  Set speed (30.0 mm/s)
  Call Extruder(0.767)
  MoveL 6356 to (509.32, 509.32, 13.5) mm, rotated rx 0 ry 90 rz 0 deg; joints [-12.669, -27.494, 110.087, -16.732, -82.041, 51.355]
  MoveL 6357 to (509.44, 509.44, 13.5) mm, rotated rx 0 ry 90 rz 0 deg; joints [-12.677, -27.491, 110.069, -16.741, -82.027, 51.361]
  Set speed (120.0 mm/s)
  MoveL 6358 to (507.39, 502.51, 13.5) mm, rotated rx 0 ry 90 rz 0 deg; joints [-12.094, -27.562, 110.499, -16.138, -82.35, 51.187]
  Set speed (30.0 mm/s)
  Call Extruder(0.280)
  MoveL 6359 to (500.58, 509.32, 13.5) mm, rotated rx 0 ry 90 rz 0 deg; joints [-12.847, -27.665, 111.134, -16.878, -82.886, 51.121]
  Set speed (120.0 mm/s)
  MoveL 6360 to (499.42, 509.32, 13.5) mm, rotated rx 0 ry 90 rz 0 deg; joints [-12.872, -27.687, 111.272, -16.898, -82.998, 51.089]
  Set speed (30.0 mm/s)
  Call Extruder(0.360)
  MoveL 6361 to (490.68, 500.58, 13.5) mm, rotated rx 0 ry 90 rz 0 deg; joints [-12.247, -27.877, 112.54, -16.235, -84.012, 50.718]
  Set speed (120.0 mm/s)
  MoveL 6362 to (490.68, 499.42, 13.5) mm, rotated rx 0 ry 90 rz 0 deg; joints [-12.139, -27.882, 112.569, -16.126, -84.034, 50.702]
  Set speed (30.0 mm/s)
  Call Extruder(0.281)
  MoveL 6363 to (497.52, 492.58, 13.5) mm, rotated rx 0 ry 90 rz 0 deg; joints [-11.373, -27.787, 111.927, -15.372, -83.486, 50.779]
  MoveL 6364 to (497.64, 492.46, 13.5) mm, rotated rx 0 ry 90 rz 0 deg; joints [-11.359, -27.786, 111.915, -15.359, -83.476, 50.78]
  Set speed (120.0 mm/s)
  MoveL 6365 to (499.02, 491.08, 13.5) mm, rotated rx 0 ry 90 rz 0 deg; joints [-11.207, -27.766, 111.784, -15.208, -83.364, 50.795]
  Set speed (30.0 mm/s)
  Call Extruder(0.016)
  MoveL 6366 to (499.42, 490.68, 13.5) mm, rotated rx 0 ry 90 rz 0 deg; joints [-11.163, -27.76, 111.745, -15.165, -83.331, 50.799]
  Set speed (120.0 mm/s)
  MoveL 6367 to (500.44, 492.33, 13.5) mm, rotated rx 0 ry 90 rz 0 deg; joints [-11.296, -27.735, 111.584, -15.303, -83.203, 50.849]
  Set speed (1000.0 mm/s)
  MoveL 6368 to (502.48, 492.58, 13.5) mm, rotated rx 0 ry 90 rz 0 deg; joints [-11.282, -27.697, 111.335, -15.296, -82.999, 50.903]
  Set speed (30.0 mm/s)
  Call Extruder(0.202)
  MoveL 6369 to (507.39, 497.49, 13.5) mm, rotated rx 0 ry 90 rz 0 deg; joints [-11.639, -27.583, 110.626, -15.676, -82.436, 51.104]
  MoveL 6370 to (507.51, 497.61, 13.5) mm, rotated rx 0 ry 90 rz 0 deg; joints [-11.648, -27.58, 110.608, -15.685, -82.422, 51.109]
  Set speed (120.0 mm/s)
  MoveL 6371 to (508.52, 498.62, 13.5) mm, rotated rx 0 ry 90 rz 0 deg; joints [-11.72, -27.556, 110.461, -15.763, -82.307, 51.151]
  Set speed (30.0 mm/s)
  Call Extruder(0.033)
  MoveL 6372 to (509.32, 499.42, 13.5) mm, rotated rx 0 ry 90 rz 0 deg; joints [-11.777, -27.537, 110.345, -15.824, -82.216, 51.185]
  Set speed (120.0 mm/s)
  MoveL 6373 to (507.64, 498.37, 13.5) mm, rotated rx 0 ry 90 rz 0 deg; joints [-11.714, -27.575, 110.573, -15.753, -82.397, 51.125]
  Set speed (1000.0 mm/s)
  MoveL 6374 to (507.64, 495.81, 13.5) mm, rotated rx 0 ry 90 rz 0 deg; joints [-11.481, -27.585, 110.637, -15.517, -82.44, 51.083]
  Set speed (1000.0 mm/s)
  MoveL 6375 to (509.32, 490.68, 13.5) mm, rotated rx 0 ry 90 rz 0 deg; joints [-10.985, -27.572, 110.557, -15.019, -82.36, 51.042]
  Set speed (30.0 mm/s)
  Call Extruder(0.767)
  MoveL 6376 to (490.68, 509.32, 13.5) mm, rotated rx 0 ry 90 rz 0 deg; joints [-13.056, -27.844, 112.308, -17.054, -83.844, 50.849]
  MoveL 6377 to (490.56, 509.44, 13.5) mm, rotated rx 0 ry 90 rz 0 deg; joints [-13.07, -27.845, 112.319, -17.068, -83.854, 50.848]
  Set speed (120.0 mm/s)
  MoveL 6378 to (502.97, 492.37, 13.5) mm, rotated rx 0 ry 90 rz 0 deg; joints [-11.253, -27.688, 111.281, -15.269, -82.954, 50.912]
  Set speed (1000.0 mm/s)
  MoveL 6379 to (502.9, 492.3, 13.5) mm, rotated rx 0 ry 90 rz 0 deg; joints [-11.248, -27.69, 111.291, -15.263, -82.962, 50.91]
  Set speed (15.0 mm/s)
  Call Extruder(0.010)
  MoveL 6380 to (502.9, 491.95, 13.5) mm, rotated rx 0 ry 90 rz 0 deg; joints [-11.216, -27.691, 111.299, -15.231, -82.968, 50.904]
  Call Extruder(0.035)
  MoveL 6381 to (502.9, 490.75, 13.5) mm, rotated rx 0 ry 90 rz 0 deg; joints [-11.106, -27.696, 111.328, -15.119, -82.988, 50.886]
  Call Extruder(0.010)
  MoveL 6382 to (502.9, 490.4, 13.5) mm, rotated rx 0 ry 90 rz 0 deg; joints [-11.074, -27.697, 111.336, -15.087, -82.994, 50.881]
  Call Extruder(0.007)
  MoveL 6383 to (503.25, 490.4, 13.5) mm, rotated rx 0 ry 90 rz 0 deg; joints [-11.068, -27.69, 111.294, -15.081, -82.96, 50.889]
  Call Extruder(0.185)
  MoveL 6384 to (509.6, 490.4, 13.5) mm, rotated rx 0 ry 90 rz 0 deg; joints [-10.955, -27.568, 110.53, -14.989, -82.337, 51.044]
  Call Extruder(0.158)
  MoveL 6385 to (509.6, 495.84, 13.5) mm, rotated rx 0 ry 90 rz 0 deg; joints [-11.448, -27.546, 110.4, -15.49, -82.249, 51.132]
  Call Extruder(0.056)
  MoveL 6386 to (507.67, 495.84, 13.5) mm, rotated rx 0 ry 90 rz 0 deg; joints [-11.483, -27.584, 110.632, -15.519, -82.437, 51.084]
  Call Extruder(0.063)
  MoveL 6387 to (507.67, 497.99, 13.5) mm, rotated rx 0 ry 90 rz 0 deg; joints [-11.679, -27.576, 110.579, -15.718, -82.4, 51.119]
  Call Extruder(0.010)
  MoveL 6388 to (507.67, 498.34, 13.5) mm, rotated rx 0 ry 90 rz 0 deg; joints [-11.711, -27.574, 110.571, -15.75, -82.394, 51.125]
  Call Extruder(0.007)
  MoveL 6389 to (508.02, 498.34, 13.5) mm, rotated rx 0 ry 90 rz 0 deg; joints [-11.704, -27.567, 110.528, -15.745, -82.36, 51.134]
  Call Extruder(0.036)
  MoveL 6390 to (509.25, 498.34, 13.5) mm, rotated rx 0 ry 90 rz 0 deg; joints [-11.681, -27.543, 110.38, -15.726, -82.241, 51.165]
  Call Extruder(0.010)
  MoveL 6391 to (509.6, 498.34, 13.5) mm, rotated rx 0 ry 90 rz 0 deg; joints [-11.675, -27.536, 110.338, -15.721, -82.206, 51.174]
  Call Extruder(0.007)
  MoveL 6392 to (509.6, 498.69, 13.5) mm, rotated rx 0 ry 90 rz 0 deg; joints [-11.706, -27.534, 110.329, -15.753, -82.201, 51.18]
  Call Extruder(0.050)
  MoveL 6393 to (509.6, 500.4, 13.5) mm, rotated rx 0 ry 90 rz 0 deg; joints [-11.86, -27.527, 110.287, -15.91, -82.171, 51.208]
  Call Extruder(0.010)
  MoveL 6394 to (509.6, 500.75, 13.5) mm, rotated rx 0 ry 90 rz 0 deg; joints [-11.892, -27.526, 110.278, -15.942, -82.165, 51.214]
  Call Extruder(0.007)
  MoveL 6395 to (509.25, 500.75, 13.5) mm, rotated rx 0 ry 90 rz 0 deg; joints [-11.898, -27.533, 110.32, -15.947, -82.199, 51.205]
  Call Extruder(0.036)
  MoveL 6396 to (508.02, 500.75, 13.5) mm, rotated rx 0 ry 90 rz 0 deg; joints [-11.922, -27.557, 110.468, -15.966, -82.319, 51.174]
  Call Extruder(0.010)
  MoveL 6397 to (507.67, 500.75, 13.5) mm, rotated rx 0 ry 90 rz 0 deg; joints [-11.928, -27.564, 110.51, -15.971, -82.353, 51.165]
  Call Extruder(0.007)
  MoveL 6398 to (507.67, 501.1, 13.5) mm, rotated rx 0 ry 90 rz 0 deg; joints [-11.96, -27.563, 110.501, -16.003, -82.347, 51.17]
  Call Extruder(0.062)
  MoveL 6399 to (507.67, 503.24, 13.5) mm, rotated rx 0 ry 90 rz 0 deg; joints [-12.154, -27.554, 110.446, -16.201, -82.31, 51.206]
  Call Extruder(0.056)
  MoveL 6400 to (509.6, 503.24, 13.5) mm, rotated rx 0 ry 90 rz 0 deg; joints [-12.117, -27.515, 110.214, -16.171, -82.122, 51.257]
  Call Extruder(0.185)
  MoveL 6401 to (509.6, 509.6, 13.5) mm, rotated rx 0 ry 90 rz 0 deg; joints [-12.688, -27.487, 110.045, -16.753, -82.009, 51.368]
  Call Extruder(0.559)
  MoveL 6402 to (490.4, 509.6, 13.5) mm, rotated rx 0 ry 90 rz 0 deg; joints [-13.088, -27.848, 112.333, -17.086, -83.866, 50.846]
  MoveL 6403 to (490.4, 490.4, 13.5) mm, rotated rx 0 ry 90 rz 0 deg; joints [-11.303, -27.917, 112.824, -15.28, -84.223, 50.569]
  Call Extruder(0.161)
  MoveL 6404 to (495.93, 490.4, 13.5) mm, rotated rx 0 ry 90 rz 0 deg; joints [-11.201, -27.823, 112.167, -15.192, -83.678, 50.708]
  Call Extruder(0.010)
  MoveL 6405 to (496.28, 490.4, 13.5) mm, rotated rx 0 ry 90 rz 0 deg; joints [-11.194, -27.817, 112.126, -15.187, -83.644, 50.717]
  Call Extruder(0.007)
  MoveL 6406 to (496.28, 490.75, 13.5) mm, rotated rx 0 ry 90 rz 0 deg; joints [-11.227, -27.816, 112.118, -15.22, -83.638, 50.722]
  Call Extruder(0.035)
  MoveL 6407 to (496.28, 491.95, 13.5) mm, rotated rx 0 ry 90 rz 0 deg; joints [-11.338, -27.812, 112.089, -15.332, -83.618, 50.739]
  Call Extruder(0.010)
  MoveL 6408 to (496.28, 492.3, 13.5) mm, rotated rx 0 ry 90 rz 0 deg; joints [-11.37, -27.81, 112.081, -15.365, -83.612, 50.744]
  Call Extruder(0.007)
  MoveL 6409 to (496.63, 492.3, 13.5) mm, rotated rx 0 ry 90 rz 0 deg; joints [-11.364, -27.804, 112.039, -15.36, -83.577, 50.753]
  Call Extruder(0.061)
  MoveL 6410 to (498.74, 492.3, 13.5) mm, rotated rx 0 ry 90 rz 0 deg; joints [-11.325, -27.767, 111.788, -15.327, -83.37, 50.806]
  Call Extruder(0.055)
  MoveL 6411 to (498.74, 490.4, 13.5) mm, rotated rx 0 ry 90 rz 0 deg; joints [-11.149, -27.773, 111.833, -15.149, -83.402, 50.778]
  Call Extruder(0.050)
  MoveL 6412 to (500.47, 490.4, 13.5) mm, rotated rx 0 ry 90 rz 0 deg; joints [-11.118, -27.742, 111.627, -15.123, -83.233, 50.821]
  Call Extruder(0.055)
  MoveL 6413 to (500.47, 492.3, 13.5) mm, rotated rx 0 ry 90 rz 0 deg; joints [-11.293, -27.735, 111.581, -15.3, -83.201, 50.849]
  Call Extruder(0.060)
  MoveL 6414 to (502.55, 492.3, 13.5) mm, rotated rx 0 ry 90 rz 0 deg; joints [-11.255, -27.696, 111.333, -15.268, -82.997, 50.901]
  Call Extruder(0.007)
  MoveL 6415 to (502.9, 492.3, 13.5) mm, rotated rx 0 ry 90 rz 0 deg; joints [-11.248, -27.69, 111.291, -15.263, -82.962, 50.91]
  Set speed (120.0 mm/s)
  MoveL 6416 to (502.9, 491.95, 13.5) mm, rotated rx 0 ry 90 rz 0 deg; joints [-11.216, -27.691, 111.299, -15.231, -82.968, 50.904]
  Set speed (1000.0 mm/s)
  MoveL 6417 to (502.9, 491.9, 13.5) mm, rotated rx 0 ry 90 rz 0 deg; joints [-11.212, -27.691, 111.3, -15.226, -82.969, 50.903]
  Set speed (1000.0 mm/s)
  MoveL 6418 to (503.6, 491.9, 13.5) mm, rotated rx 0 ry 90 rz 0 deg; joints [-11.199, -27.678, 111.216, -15.216, -82.901, 50.921]
  Set speed (1000.0 mm/s)
  MoveL 6419 to (496.25, 492.33, 13.5) mm, rotated rx 0 ry 90 rz 0 deg; joints [-11.373, -27.811, 112.083, -15.368, -83.614, 50.744]
  Set speed (1000.0 mm/s)
  MoveL 6420 to (490.68, 490.68, 13.5) mm, rotated rx 0 ry 90 rz 0 deg; joints [-11.324, -27.912, 112.784, -15.302, -84.191, 50.58]
  Set speed (1000.0 mm/s)
  MoveL 6421 to (490.68, 490.68, 13.6) mm, rotated rx 0 ry 90 rz 0 deg; joints [-11.324, -27.923, 112.789, -15.302, -84.185, 50.581]
  Set speed (30.0 mm/s)
  Call Extruder(0.767)
  MoveL 6422 to (509.32, 509.32, 13.6) mm, rotated rx 0 ry 90 rz 0 deg; joints [-12.669, -27.504, 110.092, -16.732, -82.036, 51.357]
  MoveL 6423 to (509.44, 509.44, 13.6) mm, rotated rx 0 ry 90 rz 0 deg; joints [-12.677, -27.501, 110.074, -16.741, -82.022, 51.362]
  Set speed (120.0 mm/s)
  MoveL 6424 to (507.39, 502.51, 13.6) mm, rotated rx 0 ry 90 rz 0 deg; joints [-12.094, -27.573, 110.504, -16.138, -82.345, 51.188]
  Set speed (30.0 mm/s)
  Call Extruder(0.280)
  MoveL 6425 to (500.58, 509.32, 13.6) mm, rotated rx 0 ry 90 rz 0 deg; joints [-12.847, -27.676, 111.139, -16.878, -82.88, 51.122]
  Set speed (120.0 mm/s)
  MoveL 6426 to (499.42, 509.32, 13.6) mm, rotated rx 0 ry 90 rz 0 deg; joints [-12.872, -27.698, 111.277, -16.899, -82.992, 51.091]
  Set speed (30.0 mm/s)
  Call Extruder(0.360)
  MoveL 6427 to (490.68, 500.58, 13.6) mm, rotated rx 0 ry 90 rz 0 deg; joints [-12.247, -27.888, 112.545, -16.235, -84.007, 50.72]
  Set speed (120.0 mm/s)
  MoveL 6428 to (490.68, 499.42, 13.6) mm, rotated rx 0 ry 90 rz 0 deg; joints [-12.139, -27.892, 112.575, -16.126, -84.028, 50.703]
  Set speed (30.0 mm/s)
  Call Extruder(0.281)
  MoveL 6429 to (497.52, 492.58, 13.6) mm, rotated rx 0 ry 90 rz 0 deg; joints [-11.373, -27.798, 111.932, -15.372, -83.48, 50.781]
  MoveL 6430 to (497.64, 492.46, 13.6) mm, rotated rx 0 ry 90 rz 0 deg; joints [-11.36, -27.796, 111.92, -15.359, -83.47, 50.782]
  Set speed (120.0 mm/s)
  MoveL 6431 to (498.96, 491.14, 13.6) mm, rotated rx 0 ry 90 rz 0 deg; joints [-11.213, -27.777, 111.794, -15.215, -83.363, 50.796]
  Set speed (30.0 mm/s)
  Call Extruder(0.019)
  MoveL 6432 to (499.42, 490.68, 13.6) mm, rotated rx 0 ry 90 rz 0 deg; joints [-11.163, -27.771, 111.751, -15.165, -83.326, 50.8]
  Set speed (120.0 mm/s)
  MoveL 6433 to (500.51, 492.33, 13.6) mm, rotated rx 0 ry 90 rz 0 deg; joints [-11.295, -27.745, 111.582, -15.302, -83.191, 50.852]
  Set speed (1000.0 mm/s)
  MoveL 6434 to (502.48, 492.58, 13.6) mm, rotated rx 0 ry 90 rz 0 deg; joints [-11.282, -27.707, 111.34, -15.296, -82.994, 50.905]
  Set speed (30.0 mm/s)
  Call Extruder(0.202)
  MoveL 6435 to (507.39, 497.49, 13.6) mm, rotated rx 0 ry 90 rz 0 deg; joints [-11.639, -27.594, 110.631, -15.676, -82.431, 51.105]
  MoveL 6436 to (507.51, 497.61, 13.6) mm, rotated rx 0 ry 90 rz 0 deg; joints [-11.648, -27.591, 110.613, -15.685, -82.417, 51.11]
  Set speed (120.0 mm/s)
  MoveL 6437 to (508.46, 498.57, 13.6) mm, rotated rx 0 ry 90 rz 0 deg; joints [-11.716, -27.568, 110.475, -15.759, -82.308, 51.15]
  Set speed (30.0 mm/s)
  Call Extruder(0.035)
  MoveL 6438 to (509.32, 499.42, 13.6) mm, rotated rx 0 ry 90 rz 0 deg; joints [-11.777, -27.547, 110.35, -15.824, -82.21, 51.186]
  Set speed (120.0 mm/s)
  MoveL 6439 to (507.64, 498.31, 13.6) mm, rotated rx 0 ry 90 rz 0 deg; joints [-11.709, -27.585, 110.58, -15.748, -82.392, 51.125]
  Set speed (1000.0 mm/s)
  MoveL 6440 to (507.64, 495.75, 13.6) mm, rotated rx 0 ry 90 rz 0 deg; joints [-11.476, -27.596, 110.643, -15.511, -82.436, 51.083]
  Set speed (1000.0 mm/s)
  MoveL 6441 to (509.32, 490.68, 13.6) mm, rotated rx 0 ry 90 rz 0 deg; joints [-10.985, -27.583, 110.562, -15.019, -82.355, 51.043]
  Set speed (30.0 mm/s)
  Call Extruder(0.767)
  MoveL 6442 to (490.68, 509.32, 13.6) mm, rotated rx 0 ry 90 rz 0 deg; joints [-13.056, -27.854, 112.313, -17.055, -83.839, 50.851]
  MoveL 6443 to (490.56, 509.44, 13.6) mm, rotated rx 0 ry 90 rz 0 deg; joints [-13.07, -27.856, 112.325, -17.068, -83.848, 50.849]
  Set speed (120.0 mm/s)
  MoveL 6444 to (503.03, 492.37, 13.6) mm, rotated rx 0 ry 90 rz 0 deg; joints [-11.252, -27.698, 111.278, -15.268, -82.943, 50.915]
  Set speed (1000.0 mm/s)
  MoveL 6445 to (502.96, 492.3, 13.6) mm, rotated rx 0 ry 90 rz 0 deg; joints [-11.247, -27.699, 111.288, -15.262, -82.951, 50.913]
  Set speed (15.0 mm/s)
  Call Extruder(0.010)
  MoveL 6446 to (502.96, 491.95, 13.6) mm, rotated rx 0 ry 90 rz 0 deg; joints [-11.215, -27.701, 111.297, -15.23, -82.957, 50.907]
  Call Extruder(0.035)
  MoveL 6447 to (502.96, 490.75, 13.6) mm, rotated rx 0 ry 90 rz 0 deg; joints [-11.105, -27.705, 111.325, -15.118, -82.977, 50.889]
  Call Extruder(0.010)
  MoveL 6448 to (502.96, 490.4, 13.6) mm, rotated rx 0 ry 90 rz 0 deg; joints [-11.073, -27.706, 111.333, -15.086, -82.983, 50.884]
  Call Extruder(0.007)
  MoveL 6449 to (503.31, 490.4, 13.6) mm, rotated rx 0 ry 90 rz 0 deg; joints [-11.067, -27.7, 111.291, -15.081, -82.948, 50.892]
  Call Extruder(0.183)
  MoveL 6450 to (509.6, 490.4, 13.6) mm, rotated rx 0 ry 90 rz 0 deg; joints [-10.955, -27.578, 110.535, -14.989, -82.332, 51.046]
  Call Extruder(0.156)
  MoveL 6451 to (509.6, 495.78, 13.6) mm, rotated rx 0 ry 90 rz 0 deg; joints [-11.442, -27.557, 110.407, -15.485, -82.244, 51.133]
  Call Extruder(0.056)
  MoveL 6452 to (507.67, 495.78, 13.6) mm, rotated rx 0 ry 90 rz 0 deg; joints [-11.478, -27.595, 110.639, -15.514, -82.433, 51.084]
  Call Extruder(0.063)
  MoveL 6453 to (507.67, 497.94, 13.6) mm, rotated rx 0 ry 90 rz 0 deg; joints [-11.674, -27.586, 110.586, -15.713, -82.396, 51.12]
  Call Extruder(0.010)
  MoveL 6454 to (507.67, 498.29, 13.6) mm, rotated rx 0 ry 90 rz 0 deg; joints [-11.706, -27.585, 110.577, -15.745, -82.39, 51.125]
  Call Extruder(0.007)
  MoveL 6455 to (508.02, 498.29, 13.6) mm, rotated rx 0 ry 90 rz 0 deg; joints [-11.699, -27.578, 110.535, -15.74, -82.356, 51.134]
  Call Extruder(0.036)
  MoveL 6456 to (509.25, 498.29, 13.6) mm, rotated rx 0 ry 90 rz 0 deg; joints [-11.676, -27.554, 110.387, -15.721, -82.236, 51.165]
  Call Extruder(0.010)
  MoveL 6457 to (509.6, 498.29, 13.6) mm, rotated rx 0 ry 90 rz 0 deg; joints [-11.669, -27.547, 110.345, -15.716, -82.202, 51.174]
  Call Extruder(0.007)
  MoveL 6458 to (509.6, 498.64, 13.6) mm, rotated rx 0 ry 90 rz 0 deg; joints [-11.701, -27.545, 110.336, -15.748, -82.196, 51.18]
  Call Extruder(0.053)
  MoveL 6459 to (509.6, 500.45, 13.6) mm, rotated rx 0 ry 90 rz 0 deg; joints [-11.865, -27.537, 110.29, -15.915, -82.165, 51.211]
  Call Extruder(0.010)
  MoveL 6460 to (509.6, 500.8, 13.6) mm, rotated rx 0 ry 90 rz 0 deg; joints [-11.897, -27.536, 110.281, -15.947, -82.159, 51.216]
  Call Extruder(0.007)
  MoveL 6461 to (509.25, 500.8, 13.6) mm, rotated rx 0 ry 90 rz 0 deg; joints [-11.904, -27.543, 110.324, -15.952, -82.193, 51.208]
  Call Extruder(0.036)
  MoveL 6462 to (508.02, 500.8, 13.6) mm, rotated rx 0 ry 90 rz 0 deg; joints [-11.927, -27.568, 110.472, -15.971, -82.313, 51.176]
  Call Extruder(0.010)
  MoveL 6463 to (507.67, 500.8, 13.6) mm, rotated rx 0 ry 90 rz 0 deg; joints [-11.933, -27.575, 110.514, -15.977, -82.347, 51.167]
  Call Extruder(0.007)
  MoveL 6464 to (507.67, 501.15, 13.6) mm, rotated rx 0 ry 90 rz 0 deg; joints [-11.965, -27.573, 110.505, -16.009, -82.341, 51.173]
  Call Extruder(0.062)
  MoveL 6465 to (507.67, 503.3, 13.6) mm, rotated rx 0 ry 90 rz 0 deg; joints [-12.159, -27.564, 110.45, -16.206, -82.304, 51.209]
  Call Extruder(0.056)
  MoveL 6466 to (509.6, 503.3, 13.6) mm, rotated rx 0 ry 90 rz 0 deg; joints [-12.122, -27.525, 110.217, -16.176, -82.116, 51.259]
  Call Extruder(0.183)
  MoveL 6467 to (509.6, 509.6, 13.6) mm, rotated rx 0 ry 90 rz 0 deg; joints [-12.688, -27.497, 110.05, -16.753, -82.004, 51.369]
  Call Extruder(0.559)
  MoveL 6468 to (490.4, 509.6, 13.6) mm, rotated rx 0 ry 90 rz 0 deg; joints [-13.088, -27.858, 112.339, -17.086, -83.86, 50.848]
  MoveL 6469 to (490.4, 490.4, 13.6) mm, rotated rx 0 ry 90 rz 0 deg; joints [-11.303, -27.928, 112.829, -15.28, -84.218, 50.57]
  Call Extruder(0.159)
  MoveL 6470 to (495.88, 490.4, 13.6) mm, rotated rx 0 ry 90 rz 0 deg; joints [-11.202, -27.835, 112.179, -15.193, -83.679, 50.708]
  Call Extruder(0.010)
  MoveL 6471 to (496.23, 490.4, 13.6) mm, rotated rx 0 ry 90 rz 0 deg; joints [-11.195, -27.829, 112.138, -15.188, -83.644, 50.717]
  Call Extruder(0.007)
  MoveL 6472 to (496.23, 490.75, 13.6) mm, rotated rx 0 ry 90 rz 0 deg; joints [-11.228, -27.827, 112.129, -15.221, -83.638, 50.722]
  Call Extruder(0.035)
  MoveL 6473 to (496.23, 491.95, 13.6) mm, rotated rx 0 ry 90 rz 0 deg; joints [-11.339, -27.823, 112.101, -15.333, -83.618, 50.739]
  Call Extruder(0.010)
  MoveL 6474 to (496.23, 492.3, 13.6) mm, rotated rx 0 ry 90 rz 0 deg; joints [-11.371, -27.822, 112.093, -15.366, -83.612, 50.744]
  Call Extruder(0.007)
  MoveL 6475 to (496.58, 492.3, 13.6) mm, rotated rx 0 ry 90 rz 0 deg; joints [-11.365, -27.816, 112.051, -15.361, -83.578, 50.753]
  Call Extruder(0.061)
  MoveL 6476 to (498.68, 492.3, 13.6) mm, rotated rx 0 ry 90 rz 0 deg; joints [-11.326, -27.778, 111.8, -15.328, -83.371, 50.806]
  Call Extruder(0.055)
  MoveL 6477 to (498.68, 490.4, 13.6) mm, rotated rx 0 ry 90 rz 0 deg; joints [-11.15, -27.785, 111.845, -15.15, -83.403, 50.778]
  Call Extruder(0.054)
  MoveL 6478 to (500.53, 490.4, 13.6) mm, rotated rx 0 ry 90 rz 0 deg; joints [-11.117, -27.751, 111.624, -15.122, -83.221, 50.824]
  Call Extruder(0.055)
  MoveL 6479 to (500.53, 492.3, 13.6) mm, rotated rx 0 ry 90 rz 0 deg; joints [-11.292, -27.744, 111.579, -15.299, -83.189, 50.852]
  Call Extruder(0.061)
  MoveL 6480 to (502.61, 492.3, 13.6) mm, rotated rx 0 ry 90 rz 0 deg; joints [-11.253, -27.706, 111.33, -15.268, -82.985, 50.904]
  Call Extruder(0.007)
  MoveL 6481 to (502.96, 492.3, 13.6) mm, rotated rx 0 ry 90 rz 0 deg; joints [-11.247, -27.699, 111.288, -15.262, -82.951, 50.913]
  Set speed (120.0 mm/s)
  MoveL 6482 to (502.96, 491.95, 13.6) mm, rotated rx 0 ry 90 rz 0 deg; joints [-11.215, -27.701, 111.297, -15.23, -82.957, 50.907]
  Set speed (1000.0 mm/s)
  MoveL 6483 to (502.96, 491.9, 13.6) mm, rotated rx 0 ry 90 rz 0 deg; joints [-11.21, -27.701, 111.298, -15.225, -82.958, 50.906]
  Set speed (1000.0 mm/s)
  MoveL 6484 to (503.66, 491.9, 13.6) mm, rotated rx 0 ry 90 rz 0 deg; joints [-11.198, -27.688, 111.214, -15.215, -82.889, 50.924]
  Set speed (1000.0 mm/s)
  MoveL 6485 to (496.2, 492.33, 13.6) mm, rotated rx 0 ry 90 rz 0 deg; joints [-11.374, -27.822, 112.095, -15.369, -83.614, 50.744]
  Set speed (1000.0 mm/s)
  MoveL 6486 to (490.68, 490.68, 13.6) mm, rotated rx 0 ry 90 rz 0 deg; joints [-11.324, -27.923, 112.789, -15.302, -84.185, 50.581]
  Set speed (1000.0 mm/s)
  MoveL 6487 to (490.68, 490.68, 13.7) mm, rotated rx 0 ry 90 rz 0 deg; joints [-11.324, -27.933, 112.794, -15.302, -84.18, 50.583]
  Set speed (30.0 mm/s)
  Call Extruder(0.767)
  MoveL 6488 to (509.32, 509.32, 13.7) mm, rotated rx 0 ry 90 rz 0 deg; joints [-12.669, -27.515, 110.097, -16.732, -82.031, 51.358]
  MoveL 6489 to (509.44, 509.44, 13.7) mm, rotated rx 0 ry 90 rz 0 deg; joints [-12.677, -27.511, 110.079, -16.741, -82.017, 51.364]
  Set speed (120.0 mm/s)
  MoveL 6490 to (507.39, 502.51, 13.7) mm, rotated rx 0 ry 90 rz 0 deg; joints [-12.094, -27.583, 110.509, -16.139, -82.339, 51.19]
  Set speed (30.0 mm/s)
  Call Extruder(0.280)
  MoveL 6491 to (500.58, 509.32, 13.7) mm, rotated rx 0 ry 90 rz 0 deg; joints [-12.847, -27.686, 111.144, -16.879, -82.875, 51.124]
  Set speed (120.0 mm/s)
  MoveL 6492 to (499.42, 509.32, 13.7) mm, rotated rx 0 ry 90 rz 0 deg; joints [-12.872, -27.708, 111.283, -16.899, -82.987, 51.092]
  Set speed (30.0 mm/s)
  Call Extruder(0.360)
  MoveL 6493 to (490.68, 500.58, 13.7) mm, rotated rx 0 ry 90 rz 0 deg; joints [-12.247, -27.899, 112.55, -16.235, -84.001, 50.721]
  Set speed (120.0 mm/s)
  MoveL 6494 to (490.68, 499.42, 13.7) mm, rotated rx 0 ry 90 rz 0 deg; joints [-12.139, -27.903, 112.58, -16.126, -84.023, 50.705]
  Set speed (30.0 mm/s)
  Call Extruder(0.281)
  MoveL 6495 to (497.52, 492.58, 13.7) mm, rotated rx 0 ry 90 rz 0 deg; joints [-11.373, -27.809, 111.937, -15.372, -83.475, 50.782]
  MoveL 6496 to (497.64, 492.46, 13.7) mm, rotated rx 0 ry 90 rz 0 deg; joints [-11.36, -27.807, 111.926, -15.359, -83.465, 50.783]
  Set speed (120.0 mm/s)
  MoveL 6497 to (498.91, 491.19, 13.7) mm, rotated rx 0 ry 90 rz 0 deg; joints [-11.219, -27.789, 111.805, -15.221, -83.362, 50.797]
  Set speed (30.0 mm/s)
  Call Extruder(0.021)
  MoveL 6498 to (499.42, 490.68, 13.7) mm, rotated rx 0 ry 90 rz 0 deg; joints [-11.163, -27.781, 111.756, -15.165, -83.321, 50.802]
  Set speed (120.0 mm/s)
  MoveL 6499 to (500.57, 492.33, 13.7) mm, rotated rx 0 ry 90 rz 0 deg; joints [-11.294, -27.754, 111.579, -15.302, -83.18, 50.855]
  Set speed (1000.0 mm/s)
  MoveL 6500 to (502.48, 492.58, 13.7) mm, rotated rx 0 ry 90 rz 0 deg; joints [-11.282, -27.718, 111.345, -15.296, -82.989, 50.906]
  Set speed (30.0 mm/s)
  Call Extruder(0.202)
  MoveL 6501 to (507.39, 497.49, 13.7) mm, rotated rx 0 ry 90 rz 0 deg; joints [-11.639, -27.604, 110.636, -15.676, -82.426, 51.107]
  MoveL 6502 to (507.51, 497.61, 13.7) mm, rotated rx 0 ry 90 rz 0 deg; joints [-11.648, -27.601, 110.618, -15.686, -82.412, 51.112]
  Set speed (120.0 mm/s)
  MoveL 6503 to (508.41, 498.51, 13.7) mm, rotated rx 0 ry 90 rz 0 deg; joints [-11.712, -27.58, 110.488, -15.754, -82.31, 51.149]
  Set speed (30.0 mm/s)
  Call Extruder(0.038)
  MoveL 6504 to (509.32, 499.42, 13.7) mm, rotated rx 0 ry 90 rz 0 deg; joints [-11.777, -27.558, 110.355, -15.824, -82.205, 51.187]
  Set speed (120.0 mm/s)
  MoveL 6505 to (507.64, 498.26, 13.7) mm, rotated rx 0 ry 90 rz 0 deg; joints [-11.703, -27.596, 110.586, -15.743, -82.388, 51.126]
  Set speed (1000.0 mm/s)
  MoveL 6506 to (507.64, 495.69, 13.7) mm, rotated rx 0 ry 90 rz 0 deg; joints [-11.47, -27.607, 110.65, -15.506, -82.432, 51.084]
  Set speed (1000.0 mm/s)
  MoveL 6507 to (509.32, 490.68, 13.7) mm, rotated rx 0 ry 90 rz 0 deg; joints [-10.985, -27.593, 110.568, -15.019, -82.35, 51.045]
  Set speed (30.0 mm/s)
  Call Extruder(0.767)
  MoveL 6508 to (490.68, 509.32, 13.7) mm, rotated rx 0 ry 90 rz 0 deg; joints [-13.056, -27.865, 112.319, -17.055, -83.834, 50.853]
  MoveL 6509 to (490.56, 509.44, 13.7) mm, rotated rx 0 ry 90 rz 0 deg; joints [-13.07, -27.867, 112.33, -17.068, -83.843, 50.851]
  Set speed (120.0 mm/s)
  MoveL 6510 to (503.1, 492.37, 13.7) mm, rotated rx 0 ry 90 rz 0 deg; joints [-11.251, -27.707, 111.276, -15.267, -82.931, 50.918]
  Set speed (1000.0 mm/s)
  MoveL 6511 to (503.03, 492.3, 13.7) mm, rotated rx 0 ry 90 rz 0 deg; joints [-11.246, -27.709, 111.286, -15.262, -82.94, 50.916]
  Set speed (15.0 mm/s)
  Call Extruder(0.010)
  MoveL 6512 to (503.03, 491.95, 13.7) mm, rotated rx 0 ry 90 rz 0 deg; joints [-11.214, -27.71, 111.294, -15.229, -82.945, 50.91]
  Call Extruder(0.035)
  MoveL 6513 to (503.03, 490.75, 13.7) mm, rotated rx 0 ry 90 rz 0 deg; joints [-11.104, -27.714, 111.323, -15.118, -82.965, 50.892]
  Call Extruder(0.010)
  MoveL 6514 to (503.03, 490.4, 13.7) mm, rotated rx 0 ry 90 rz 0 deg; joints [-11.072, -27.716, 111.331, -15.085, -82.971, 50.887]
  Call Extruder(0.007)
  MoveL 6515 to (503.38, 490.4, 13.7) mm, rotated rx 0 ry 90 rz 0 deg; joints [-11.065, -27.709, 111.289, -15.08, -82.937, 50.895]
  Call Extruder(0.181)
  MoveL 6516 to (509.6, 490.4, 13.7) mm, rotated rx 0 ry 90 rz 0 deg; joints [-10.955, -27.589, 110.54, -14.989, -82.327, 51.047]
  Call Extruder(0.155)
  MoveL 6517 to (509.6, 495.71, 13.7) mm, rotated rx 0 ry 90 rz 0 deg; joints [-11.437, -27.568, 110.413, -15.479, -82.24, 51.133]
  Call Extruder(0.056)
  MoveL 6518 to (507.67, 495.72, 13.7) mm, rotated rx 0 ry 90 rz 0 deg; joints [-11.473, -27.606, 110.646, -15.508, -82.428, 51.085]
  Call Extruder(0.063)
  MoveL 6519 to (507.67, 497.88, 13.7) mm, rotated rx 0 ry 90 rz 0 deg; joints [-11.668, -27.597, 110.592, -15.707, -82.392, 51.12]
  Call Extruder(0.010)
  MoveL 6520 to (507.67, 498.23, 13.7) mm, rotated rx 0 ry 90 rz 0 deg; joints [-11.7, -27.596, 110.584, -15.74, -82.386, 51.126]
  Call Extruder(0.007)
  MoveL 6521 to (508.02, 498.23, 13.7) mm, rotated rx 0 ry 90 rz 0 deg; joints [-11.694, -27.589, 110.542, -15.734, -82.352, 51.135]
  Call Extruder(0.036)
  MoveL 6522 to (509.25, 498.23, 13.7) mm, rotated rx 0 ry 90 rz 0 deg; joints [-11.671, -27.564, 110.394, -15.716, -82.232, 51.166]
  Call Extruder(0.010)
  MoveL 6523 to (509.6, 498.23, 13.7) mm, rotated rx 0 ry 90 rz 0 deg; joints [-11.664, -27.557, 110.351, -15.71, -82.198, 51.175]
  Call Extruder(0.007)
  MoveL 6524 to (509.6, 498.58, 13.7) mm, rotated rx 0 ry 90 rz 0 deg; joints [-11.696, -27.556, 110.343, -15.743, -82.192, 51.18]
  Call Extruder(0.056)
  MoveL 6525 to (509.6, 500.51, 13.7) mm, rotated rx 0 ry 90 rz 0 deg; joints [-11.87, -27.548, 110.294, -15.92, -82.159, 51.213]
  Call Extruder(0.010)
  MoveL 6526 to (509.6, 500.86, 13.7) mm, rotated rx 0 ry 90 rz 0 deg; joints [-11.902, -27.546, 110.285, -15.952, -82.153, 51.219]
  Call Extruder(0.007)
  MoveL 6527 to (509.25, 500.86, 13.7) mm, rotated rx 0 ry 90 rz 0 deg; joints [-11.909, -27.553, 110.327, -15.958, -82.187, 51.21]
  Call Extruder(0.036)
  MoveL 6528 to (508.02, 500.86, 13.7) mm, rotated rx 0 ry 90 rz 0 deg; joints [-11.932, -27.578, 110.476, -15.977, -82.307, 51.178]
  Call Extruder(0.010)
  MoveL 6529 to (507.67, 500.86, 13.7) mm, rotated rx 0 ry 90 rz 0 deg; joints [-11.939, -27.585, 110.518, -15.982, -82.341, 51.17]
  Call Extruder(0.007)
  MoveL 6530 to (507.67, 501.21, 13.7) mm, rotated rx 0 ry 90 rz 0 deg; joints [-11.97, -27.583, 110.509, -16.014, -82.335, 51.175]
  Call Extruder(0.062)
  MoveL 6531 to (507.67, 503.35, 13.7) mm, rotated rx 0 ry 90 rz 0 deg; joints [-12.164, -27.574, 110.454, -16.211, -82.297, 51.211]
  Call Extruder(0.056)
  MoveL 6532 to (509.6, 503.36, 13.7) mm, rotated rx 0 ry 90 rz 0 deg; joints [-12.127, -27.535, 110.221, -16.181, -82.11, 51.261]
  Call Extruder(0.182)
  MoveL 6533 to (509.6, 509.6, 13.7) mm, rotated rx 0 ry 90 rz 0 deg; joints [-12.688, -27.508, 110.056, -16.753, -81.998, 51.371]
  Call Extruder(0.559)
  MoveL 6534 to (490.4, 509.6, 13.7) mm, rotated rx 0 ry 90 rz 0 deg; joints [-13.088, -27.869, 112.344, -17.086, -83.855, 50.849]
  MoveL 6535 to (490.4, 490.4, 13.7) mm, rotated rx 0 ry 90 rz 0 deg; joints [-11.303, -27.939, 112.834, -15.28, -84.212, 50.572]
  Call Extruder(0.168)
  MoveL 6536 to (496.17, 490.4, 13.7) mm, rotated rx 0 ry 90 rz 0 deg; joints [-11.196, -27.84, 112.15, -15.189, -83.645, 50.717]
  Call Extruder(0.055)
  MoveL 6537 to (496.17, 492.3, 13.7) mm, rotated rx 0 ry 90 rz 0 deg; joints [-11.372, -27.834, 112.104, -15.367, -83.612, 50.744]
  Call Extruder(0.071)
  MoveL 6538 to (498.63, 492.3, 13.7) mm, rotated rx 0 ry 90 rz 0 deg; joints [-11.327, -27.79, 111.812, -15.329, -83.371, 50.806]
  Call Extruder(0.055)
  MoveL 6539 to (498.63, 490.4, 13.7) mm, rotated rx 0 ry 90 rz 0 deg; joints [-11.151, -27.797, 111.857, -15.151, -83.403, 50.778]
  Call Extruder(0.057)
  MoveL 6540 to (500.6, 490.4, 13.7) mm, rotated rx 0 ry 90 rz 0 deg; joints [-11.115, -27.761, 111.622, -15.121, -83.21, 50.827]
  Call Extruder(0.055)
  MoveL 6541 to (500.6, 492.3, 13.7) mm, rotated rx 0 ry 90 rz 0 deg; joints [-11.29, -27.754, 111.577, -15.299, -83.178, 50.855]
  Call Extruder(0.061)
  MoveL 6542 to (502.68, 492.3, 13.7) mm, rotated rx 0 ry 90 rz 0 deg; joints [-11.252, -27.715, 111.328, -15.267, -82.974, 50.907]
  Call Extruder(0.007)
  MoveL 6543 to (503.03, 492.3, 13.7) mm, rotated rx 0 ry 90 rz 0 deg; joints [-11.246, -27.709, 111.286, -15.262, -82.94, 50.916]
  Set speed (120.0 mm/s)
  MoveL 6544 to (503.03, 491.95, 13.7) mm, rotated rx 0 ry 90 rz 0 deg; joints [-11.214, -27.71, 111.294, -15.229, -82.945, 50.91]
  Set speed (1000.0 mm/s)
  MoveL 6545 to (503.03, 491.9, 13.7) mm, rotated rx 0 ry 90 rz 0 deg; joints [-11.209, -27.71, 111.295, -15.224, -82.946, 50.909]
  Set speed (1000.0 mm/s)
  MoveL 6546 to (503.73, 491.9, 13.7) mm, rotated rx 0 ry 90 rz 0 deg; joints [-11.197, -27.697, 111.211, -15.214, -82.878, 50.927]
  Set speed (1000.0 mm/s)
  MoveL 6547 to (496.14, 492.33, 13.7) mm, rotated rx 0 ry 90 rz 0 deg; joints [-11.375, -27.834, 112.107, -15.37, -83.614, 50.744]
  Set speed (1000.0 mm/s)
  MoveL 6548 to (490.68, 490.68, 13.7) mm, rotated rx 0 ry 90 rz 0 deg; joints [-11.324, -27.933, 112.794, -15.302, -84.18, 50.583]
  Set speed (1000.0 mm/s)
  MoveL 6549 to (490.68, 490.68, 13.8) mm, rotated rx 0 ry 90 rz 0 deg; joints [-11.324, -27.944, 112.8, -15.302, -84.175, 50.584]
  Set speed (30.0 mm/s)
  Call Extruder(0.767)
  MoveL 6550 to (509.32, 509.32, 13.8) mm, rotated rx 0 ry 90 rz 0 deg; joints [-12.669, -27.525, 110.102, -16.732, -82.026, 51.36]
  MoveL 6551 to (509.44, 509.44, 13.8) mm, rotated rx 0 ry 90 rz 0 deg; joints [-12.677, -27.522, 110.084, -16.741, -82.011, 51.365]
  Set speed (120.0 mm/s)
  MoveL 6552 to (507.39, 502.51, 13.8) mm, rotated rx 0 ry 90 rz 0 deg; joints [-12.094, -27.594, 110.514, -16.139, -82.334, 51.191]
  Set speed (30.0 mm/s)
  Call Extruder(0.280)
  MoveL 6553 to (500.58, 509.32, 13.8) mm, rotated rx 0 ry 90 rz 0 deg; joints [-12.847, -27.697, 111.15, -16.879, -82.87, 51.125]
  Set speed (120.0 mm/s)
  MoveL 6554 to (499.42, 509.32, 13.8) mm, rotated rx 0 ry 90 rz 0 deg; joints [-12.872, -27.719, 111.288, -16.899, -82.982, 51.094]
  Set speed (30.0 mm/s)
  Call Extruder(0.360)
  MoveL 6555 to (490.68, 500.58, 13.8) mm, rotated rx 0 ry 90 rz 0 deg; joints [-12.247, -27.909, 112.555, -16.235, -83.996, 50.723]
  Set speed (120.0 mm/s)
  MoveL 6556 to (490.68, 499.42, 13.8) mm, rotated rx 0 ry 90 rz 0 deg; joints [-12.139, -27.914, 112.585, -16.126, -84.018, 50.706]
  Set speed (30.0 mm/s)
  Call Extruder(0.281)
  MoveL 6557 to (497.52, 492.58, 13.8) mm, rotated rx 0 ry 90 rz 0 deg; joints [-11.373, -27.819, 111.942, -15.373, -83.47, 50.784]
  MoveL 6558 to (497.64, 492.46, 13.8) mm, rotated rx 0 ry 90 rz 0 deg; joints [-11.36, -27.818, 111.931, -15.359, -83.46, 50.785]
  Set speed (120.0 mm/s)
  MoveL 6559 to (498.85, 491.25, 13.8) mm, rotated rx 0 ry 90 rz 0 deg; joints [-11.226, -27.8, 111.815, -15.227, -83.362, 50.797]
  Set speed (30.0 mm/s)
  Call Extruder(0.023)
  MoveL 6560 to (499.42, 490.68, 13.8) mm, rotated rx 0 ry 90 rz 0 deg; joints [-11.163, -27.792, 111.761, -15.165, -83.315, 50.803]
  Set speed (120.0 mm/s)
  MoveL 6561 to (500.63, 492.33, 13.8) mm, rotated rx 0 ry 90 rz 0 deg; joints [-11.292, -27.764, 111.577, -15.301, -83.169, 50.858]
  Set speed (1000.0 mm/s)
  MoveL 6562 to (502.48, 492.58, 13.8) mm, rotated rx 0 ry 90 rz 0 deg; joints [-11.282, -27.728, 111.35, -15.296, -82.983, 50.908]
  Set speed (30.0 mm/s)
  Call Extruder(0.202)
  MoveL 6563 to (507.39, 497.49, 13.8) mm, rotated rx 0 ry 90 rz 0 deg; joints [-11.639, -27.615, 110.641, -15.676, -82.421, 51.108]
  Set speed (120.0 mm/s)
  MoveL 6564 to (508.35, 498.45, 13.8) mm, rotated rx 0 ry 90 rz 0 deg; joints [-11.708, -27.592, 110.502, -15.75, -82.311, 51.148]
  Set speed (30.0 mm/s)
  Call Extruder(0.040)
  MoveL 6565 to (509.32, 499.42, 13.8) mm, rotated rx 0 ry 90 rz 0 deg; joints [-11.777, -27.568, 110.36, -15.825, -82.2, 51.189]
  Set speed (120.0 mm/s)
  MoveL 6566 to (507.64, 498.2, 13.8) mm, rotated rx 0 ry 90 rz 0 deg; joints [-11.698, -27.607, 110.593, -15.738, -82.384, 51.126]
  Set speed (1000.0 mm/s)
  MoveL 6567 to (507.64, 495.63, 13.8) mm, rotated rx 0 ry 90 rz 0 deg; joints [-11.465, -27.617, 110.656, -15.501, -82.427, 51.084]
  Set speed (1000.0 mm/s)
  MoveL 6568 to (509.32, 490.68, 13.8) mm, rotated rx 0 ry 90 rz 0 deg; joints [-10.985, -27.604, 110.573, -15.019, -82.345, 51.046]
  Set speed (30.0 mm/s)
  Call Extruder(0.767)
  MoveL 6569 to (490.68, 509.32, 13.8) mm, rotated rx 0 ry 90 rz 0 deg; joints [-13.056, -27.876, 112.324, -17.055, -83.828, 50.854]
  MoveL 6570 to (490.56, 509.44, 13.8) mm, rotated rx 0 ry 90 rz 0 deg; joints [-13.07, -27.877, 112.335, -17.069, -83.838, 50.853]
  Set speed (120.0 mm/s)
  MoveL 6571 to (503.16, 492.37, 13.8) mm, rotated rx 0 ry 90 rz 0 deg; joints [-11.25, -27.716, 111.273, -15.266, -82.92, 50.921]
  Set speed (1000.0 mm/s)
  MoveL 6572 to (503.09, 492.3, 13.8) mm, rotated rx 0 ry 90 rz 0 deg; joints [-11.245, -27.718, 111.283, -15.261, -82.928, 50.919]
  Set speed (15.0 mm/s)
  Call Extruder(0.010)
  MoveL 6573 to (503.09, 491.95, 13.8) mm, rotated rx 0 ry 90 rz 0 deg; joints [-11.213, -27.719, 111.292, -15.228, -82.934, 50.913]
  Call Extruder(0.035)
  MoveL 6574 to (503.09, 490.75, 13.8) mm, rotated rx 0 ry 90 rz 0 deg; joints [-11.103, -27.724, 111.32, -15.117, -82.954, 50.895]
  Call Extruder(0.010)
  MoveL 6575 to (503.09, 490.4, 13.8) mm, rotated rx 0 ry 90 rz 0 deg; joints [-11.071, -27.725, 111.328, -15.084, -82.96, 50.89]
  Call Extruder(0.007)
  MoveL 6576 to (503.44, 490.4, 13.8) mm, rotated rx 0 ry 90 rz 0 deg; joints [-11.064, -27.718, 111.286, -15.079, -82.925, 50.898]
  Call Extruder(0.179)
  MoveL 6577 to (509.6, 490.4, 13.8) mm, rotated rx 0 ry 90 rz 0 deg; joints [-10.955, -27.599, 110.545, -14.99, -82.322, 51.048]
  Call Extruder(0.153)
  MoveL 6578 to (509.6, 495.66, 13.8) mm, rotated rx 0 ry 90 rz 0 deg; joints [-11.432, -27.578, 110.42, -15.474, -82.236, 51.134]
  Call Extruder(0.056)
  MoveL 6579 to (507.67, 495.66, 13.8) mm, rotated rx 0 ry 90 rz 0 deg; joints [-11.467, -27.617, 110.652, -15.503, -82.424, 51.085]
  Call Extruder(0.063)
  MoveL 6580 to (507.67, 497.82, 13.8) mm, rotated rx 0 ry 90 rz 0 deg; joints [-11.663, -27.608, 110.599, -15.702, -82.388, 51.121]
  Call Extruder(0.010)
  MoveL 6581 to (507.67, 498.17, 13.8) mm, rotated rx 0 ry 90 rz 0 deg; joints [-11.695, -27.606, 110.59, -15.735, -82.382, 51.126]
  Call Extruder(0.007)
  MoveL 6582 to (508.02, 498.17, 13.8) mm, rotated rx 0 ry 90 rz 0 deg; joints [-11.688, -27.6, 110.548, -15.729, -82.348, 51.135]
  Call Extruder(0.036)
  MoveL 6583 to (509.25, 498.17, 13.8) mm, rotated rx 0 ry 90 rz 0 deg; joints [-11.665, -27.575, 110.4, -15.71, -82.228, 51.166]
  Call Extruder(0.010)
  MoveL 6584 to (509.6, 498.17, 13.8) mm, rotated rx 0 ry 90 rz 0 deg; joints [-11.659, -27.568, 110.358, -15.705, -82.194, 51.175]
  Call Extruder(0.007)
  MoveL 6585 to (509.6, 498.52, 13.8) mm, rotated rx 0 ry 90 rz 0 deg; joints [-11.69, -27.567, 110.349, -15.737, -82.188, 51.181]
  Call Extruder(0.060)
  MoveL 6586 to (509.6, 500.57, 13.8) mm, rotated rx 0 ry 90 rz 0 deg; joints [-11.875, -27.558, 110.298, -15.925, -82.153, 51.215]
  Call Extruder(0.010)
  MoveL 6587 to (509.6, 500.92, 13.8) mm, rotated rx 0 ry 90 rz 0 deg; joints [-11.907, -27.556, 110.289, -15.958, -82.147, 51.221]
  Call Extruder(0.007)
  MoveL 6588 to (509.25, 500.92, 13.8) mm, rotated rx 0 ry 90 rz 0 deg; joints [-11.914, -27.563, 110.331, -15.963, -82.181, 51.212]
  Call Extruder(0.036)
  MoveL 6589 to (508.02, 500.91, 13.8) mm, rotated rx 0 ry 90 rz 0 deg; joints [-11.937, -27.588, 110.479, -15.982, -82.301, 51.181]
  Call Extruder(0.010)
  MoveL 6590 to (507.67, 500.91, 13.8) mm, rotated rx 0 ry 90 rz 0 deg; joints [-11.943, -27.595, 110.521, -15.987, -82.335, 51.172]
  Call Extruder(0.007)
  MoveL 6591 to (507.67, 501.26, 13.8) mm, rotated rx 0 ry 90 rz 0 deg; joints [-11.975, -27.594, 110.513, -16.019, -82.329, 51.178]
  Call Extruder(0.062)
  MoveL 6592 to (507.67, 503.41, 13.8) mm, rotated rx 0 ry 90 rz 0 deg; joints [-12.169, -27.585, 110.457, -16.217, -82.291, 51.214]
  Call Extruder(0.056)
  MoveL 6593 to (509.6, 503.41, 13.8) mm, rotated rx 0 ry 90 rz 0 deg; joints [-12.132, -27.546, 110.225, -16.187, -82.104, 51.264]
  Call Extruder(0.180)
  MoveL 6594 to (509.6, 509.6, 13.8) mm, rotated rx 0 ry 90 rz 0 deg; joints [-12.688, -27.518, 110.061, -16.753, -81.993, 51.372]
  Call Extruder(0.559)
  MoveL 6595 to (490.4, 509.6, 13.8) mm, rotated rx 0 ry 90 rz 0 deg; joints [-13.088, -27.879, 112.349, -17.086, -83.85, 50.851]
  MoveL 6596 to (490.4, 490.4, 13.8) mm, rotated rx 0 ry 90 rz 0 deg; joints [-11.303, -27.95, 112.839, -15.28, -84.207, 50.573]
  Call Extruder(0.156)
  MoveL 6597 to (495.76, 490.4, 13.8) mm, rotated rx 0 ry 90 rz 0 deg; joints [-11.204, -27.858, 112.203, -15.195, -83.679, 50.708]
  Call Extruder(0.010)
  MoveL 6598 to (496.11, 490.4, 13.8) mm, rotated rx 0 ry 90 rz 0 deg; joints [-11.197, -27.852, 112.161, -15.19, -83.645, 50.717]
  Call Extruder(0.007)
  MoveL 6599 to (496.11, 490.75, 13.8) mm, rotated rx 0 ry 90 rz 0 deg; joints [-11.23, -27.851, 112.153, -15.223, -83.639, 50.722]
  Call Extruder(0.035)
  MoveL 6600 to (496.11, 491.95, 13.8) mm, rotated rx 0 ry 90 rz 0 deg; joints [-11.341, -27.846, 112.125, -15.336, -83.618, 50.739]
  Call Extruder(0.010)
  MoveL 6601 to (496.11, 492.3, 13.8) mm, rotated rx 0 ry 90 rz 0 deg; joints [-11.373, -27.845, 112.116, -15.368, -83.612, 50.744]
  Call Extruder(0.007)
  MoveL 6602 to (496.46, 492.3, 13.8) mm, rotated rx 0 ry 90 rz 0 deg; joints [-11.367, -27.839, 112.075, -15.363, -83.578, 50.753]
  Call Extruder(0.061)
  MoveL 6603 to (498.57, 492.3, 13.8) mm, rotated rx 0 ry 90 rz 0 deg; joints [-11.328, -27.801, 111.824, -15.33, -83.371, 50.806]
  Call Extruder(0.055)
  MoveL 6604 to (498.57, 490.4, 13.8) mm, rotated rx 0 ry 90 rz 0 deg; joints [-11.152, -27.808, 111.869, -15.152, -83.403, 50.778]
  Call Extruder(0.061)
  MoveL 6605 to (500.66, 490.4, 13.8) mm, rotated rx 0 ry 90 rz 0 deg; joints [-11.114, -27.77, 111.619, -15.121, -83.198, 50.83]
  Call Extruder(0.055)
  MoveL 6606 to (500.66, 492.3, 13.8) mm, rotated rx 0 ry 90 rz 0 deg; joints [-11.289, -27.763, 111.574, -15.298, -83.166, 50.858]
  Call Extruder(0.061)
  MoveL 6607 to (502.74, 492.3, 13.8) mm, rotated rx 0 ry 90 rz 0 deg; joints [-11.251, -27.725, 111.325, -15.266, -82.962, 50.91]
  Call Extruder(0.007)
  MoveL 6608 to (503.09, 492.3, 13.8) mm, rotated rx 0 ry 90 rz 0 deg; joints [-11.245, -27.718, 111.283, -15.261, -82.928, 50.919]
  Set speed (120.0 mm/s)
  MoveL 6609 to (503.09, 491.95, 13.8) mm, rotated rx 0 ry 90 rz 0 deg; joints [-11.213, -27.719, 111.292, -15.228, -82.934, 50.913]
  Set speed (1000.0 mm/s)
  MoveL 6610 to (503.09, 491.9, 13.8) mm, rotated rx 0 ry 90 rz 0 deg; joints [-11.208, -27.719, 111.293, -15.224, -82.935, 50.912]
  Set speed (1000.0 mm/s)
  MoveL 6611 to (503.79, 491.9, 13.8) mm, rotated rx 0 ry 90 rz 0 deg; joints [-11.195, -27.706, 111.209, -15.213, -82.866, 50.93]
  Set speed (1000.0 mm/s)
  MoveL 6612 to (496.08, 492.33, 13.8) mm, rotated rx 0 ry 90 rz 0 deg; joints [-11.377, -27.846, 112.119, -15.371, -83.615, 50.744]
  Set speed (1000.0 mm/s)
  MoveL 6613 to (490.68, 490.68, 13.8) mm, rotated rx 0 ry 90 rz 0 deg; joints [-11.324, -27.944, 112.8, -15.302, -84.175, 50.584]
  Set speed (1000.0 mm/s)
  MoveL 6614 to (490.68, 490.68, 13.9) mm, rotated rx 0 ry 90 rz 0 deg; joints [-11.324, -27.955, 112.805, -15.302, -84.169, 50.586]
  Set speed (30.0 mm/s)
  Call Extruder(0.767)
  MoveL 6615 to (509.32, 509.32, 13.9) mm, rotated rx 0 ry 90 rz 0 deg; joints [-12.669, -27.535, 110.107, -16.732, -82.02, 51.361]
  MoveL 6616 to (509.44, 509.44, 13.9) mm, rotated rx 0 ry 90 rz 0 deg; joints [-12.677, -27.532, 110.089, -16.742, -82.006, 51.367]
  Set speed (120.0 mm/s)
  MoveL 6617 to (508.42, 506.07, 13.9) mm, rotated rx 0 ry 90 rz 0 deg; joints [-12.394, -27.568, 110.302, -16.449, -82.166, 51.281]
  Set speed (1000.0 mm/s)
  MoveL 6618 to (507.39, 502.51, 13.9) mm, rotated rx 0 ry 90 rz 0 deg; joints [-12.094, -27.604, 110.52, -16.139, -82.329, 51.193]
  Set speed (30.0 mm/s)
  Call Extruder(0.280)
  MoveL 6619 to (500.58, 509.32, 13.9) mm, rotated rx 0 ry 90 rz 0 deg; joints [-12.847, -27.707, 111.155, -16.879, -82.865, 51.127]
  Set speed (120.0 mm/s)
  MoveL 6620 to (499.42, 509.32, 13.9) mm, rotated rx 0 ry 90 rz 0 deg; joints [-12.872, -27.729, 111.293, -16.899, -82.977, 51.096]
  Set speed (30.0 mm/s)
  Call Extruder(0.360)
  MoveL 6621 to (490.68, 500.58, 13.9) mm, rotated rx 0 ry 90 rz 0 deg; joints [-12.247, -27.92, 112.561, -16.235, -83.991, 50.725]
  Set speed (120.0 mm/s)
  MoveL 6622 to (490.68, 499.42, 13.9) mm, rotated rx 0 ry 90 rz 0 deg; joints [-12.139, -27.924, 112.59, -16.126, -84.012, 50.708]
  Set speed (30.0 mm/s)
  Call Extruder(0.281)
  MoveL 6623 to (497.52, 492.58, 13.9) mm, rotated rx 0 ry 90 rz 0 deg; joints [-11.373, -27.83, 111.948, -15.373, -83.464, 50.785]
  MoveL 6624 to (497.64, 492.46, 13.9) mm, rotated rx 0 ry 90 rz 0 deg; joints [-11.36, -27.828, 111.936, -15.359, -83.455, 50.786]
  Set speed (120.0 mm/s)
  MoveL 6625 to (498.79, 491.31, 13.9) mm, rotated rx 0 ry 90 rz 0 deg; joints [-11.232, -27.812, 111.826, -15.234, -83.361, 50.798]
  Set speed (30.0 mm/s)
  Call Extruder(0.026)
  MoveL 6626 to (499.42, 490.68, 13.9) mm, rotated rx 0 ry 90 rz 0 deg; joints [-11.163, -27.802, 111.766, -15.166, -83.31, 50.805]
  Set speed (120.0 mm/s)
  MoveL 6627 to (500.7, 492.33, 13.9) mm, rotated rx 0 ry 90 rz 0 deg; joints [-11.291, -27.773, 111.574, -15.3, -83.157, 50.861]
  Set speed (1000.0 mm/s)
  MoveL 6628 to (502.48, 492.58, 13.9) mm, rotated rx 0 ry 90 rz 0 deg; joints [-11.282, -27.739, 111.355, -15.296, -82.978, 50.909]
  Set speed (30.0 mm/s)
  Call Extruder(0.202)
  MoveL 6629 to (507.39, 497.49, 13.9) mm, rotated rx 0 ry 90 rz 0 deg; joints [-11.639, -27.625, 110.646, -15.677, -82.416, 51.11]
  Set speed (120.0 mm/s)
  MoveL 6630 to (508.29, 498.39, 13.9) mm, rotated rx 0 ry 90 rz 0 deg; joints [-11.703, -27.604, 110.515, -15.746, -82.313, 51.147]
  Set speed (30.0 mm/s)
  Call Extruder(0.042)
  MoveL 6631 to (509.32, 499.42, 13.9) mm, rotated rx 0 ry 90 rz 0 deg; joints [-11.777, -27.579, 110.366, -15.825, -82.195, 51.19]
  Set speed (120.0 mm/s)
  MoveL 6632 to (509.32, 500.58, 13.9) mm, rotated rx 0 ry 90 rz 0 deg; joints [-11.882, -27.574, 110.336, -15.931, -82.175, 51.21]
  Set speed (30.0 mm/s)
  Call Extruder(0.005)
  MoveL 6633 to (509.21, 500.69, 13.9) mm, rotated rx 0 ry 90 rz 0 deg; joints [-11.894, -27.576, 110.347, -15.943, -82.184, 51.209]
  Set speed (120.0 mm/s)
  MoveL 6634 to (507.64, 498.14, 13.9) mm, rotated rx 0 ry 90 rz 0 deg; joints [-11.693, -27.618, 110.6, -15.732, -82.38, 51.127]
  Set speed (1000.0 mm/s)
  MoveL 6635 to (507.64, 495.57, 13.9) mm, rotated rx 0 ry 90 rz 0 deg; joints [-11.46, -27.628, 110.663, -15.496, -82.423, 51.085]
  Set speed (1000.0 mm/s)
  MoveL 6636 to (509.32, 490.68, 13.9) mm, rotated rx 0 ry 90 rz 0 deg; joints [-10.985, -27.614, 110.578, -15.02, -82.339, 51.047]
  Set speed (30.0 mm/s)
  Call Extruder(0.767)
  MoveL 6637 to (490.68, 509.32, 13.9) mm, rotated rx 0 ry 90 rz 0 deg; joints [-13.056, -27.886, 112.329, -17.055, -83.823, 50.856]
  MoveL 6638 to (490.56, 509.44, 13.9) mm, rotated rx 0 ry 90 rz 0 deg; joints [-13.07, -27.888, 112.34, -17.069, -83.833, 50.854]
  Set speed (120.0 mm/s)
  MoveL 6639 to (503.22, 492.37, 13.9) mm, rotated rx 0 ry 90 rz 0 deg; joints [-11.249, -27.726, 111.271, -15.266, -82.909, 50.924]
  Set speed (1000.0 mm/s)
  MoveL 6640 to (503.15, 492.3, 13.9) mm, rotated rx 0 ry 90 rz 0 deg; joints [-11.244, -27.727, 111.281, -15.26, -82.917, 50.922]
  Set speed (15.0 mm/s)
  Call Extruder(0.010)
  MoveL 6641 to (503.15, 491.95, 13.9) mm, rotated rx 0 ry 90 rz 0 deg; joints [-11.211, -27.729, 111.289, -15.228, -82.922, 50.916]
  Call Extruder(0.035)
  MoveL 6642 to (503.15, 490.75, 13.9) mm, rotated rx 0 ry 90 rz 0 deg; joints [-11.101, -27.733, 111.318, -15.116, -82.942, 50.898]
  Call Extruder(0.010)
  MoveL 6643 to (503.15, 490.4, 13.9) mm, rotated rx 0 ry 90 rz 0 deg; joints [-11.069, -27.734, 111.326, -15.083, -82.948, 50.893]
  Call Extruder(0.007)
  MoveL 6644 to (503.5, 490.4, 13.9) mm, rotated rx 0 ry 90 rz 0 deg; joints [-11.063, -27.728, 111.284, -15.078, -82.914, 50.901]
  Call Extruder(0.177)
  MoveL 6645 to (509.6, 490.4, 13.9) mm, rotated rx 0 ry 90 rz 0 deg; joints [-10.955, -27.61, 110.55, -14.99, -82.316, 51.05]
  Call Extruder(0.151)
  MoveL 6646 to (509.6, 495.6, 13.9) mm, rotated rx 0 ry 90 rz 0 deg; joints [-11.426, -27.589, 110.426, -15.469, -82.232, 51.134]
  Call Extruder(0.056)
  MoveL 6647 to (507.67, 495.6, 13.9) mm, rotated rx 0 ry 90 rz 0 deg; joints [-11.462, -27.627, 110.659, -15.498, -82.42, 51.086]
  Call Extruder(0.063)
  MoveL 6648 to (507.67, 497.76, 13.9) mm, rotated rx 0 ry 90 rz 0 deg; joints [-11.658, -27.619, 110.606, -15.697, -82.384, 51.121]
  Call Extruder(0.010)
  MoveL 6649 to (507.67, 498.11, 13.9) mm, rotated rx 0 ry 90 rz 0 deg; joints [-11.69, -27.617, 110.597, -15.729, -82.378, 51.127]
  Call Extruder(0.007)
  MoveL 6650 to (508.02, 498.11, 13.9) mm, rotated rx 0 ry 90 rz 0 deg; joints [-11.683, -27.61, 110.555, -15.724, -82.344, 51.136]
  Call Extruder(0.046)
  MoveL 6651 to (509.6, 498.11, 13.9) mm, rotated rx 0 ry 90 rz 0 deg; joints [-11.653, -27.579, 110.364, -15.7, -82.19, 51.176]
  Call Extruder(0.083)
  MoveL 6652 to (509.6, 500.97, 13.9) mm, rotated rx 0 ry 90 rz 0 deg; joints [-11.912, -27.567, 110.292, -15.963, -82.141, 51.224]
  Call Extruder(0.046)
  MoveL 6653 to (508.02, 500.97, 13.9) mm, rotated rx 0 ry 90 rz 0 deg; joints [-11.942, -27.598, 110.483, -15.987, -82.295, 51.183]
  Call Extruder(0.010)
  MoveL 6654 to (507.67, 500.97, 13.9) mm, rotated rx 0 ry 90 rz 0 deg; joints [-11.949, -27.605, 110.525, -15.993, -82.329, 51.174]
  Call Extruder(0.007)
  MoveL 6655 to (507.67, 501.32, 13.9) mm, rotated rx 0 ry 90 rz 0 deg; joints [-11.98, -27.604, 110.516, -16.025, -82.323, 51.18]
  Call Extruder(0.062)
  MoveL 6656 to (507.67, 503.46, 13.9) mm, rotated rx 0 ry 90 rz 0 deg; joints [-12.174, -27.595, 110.461, -16.222, -82.285, 51.216]
  Call Extruder(0.056)
  MoveL 6657 to (509.6, 503.47, 13.9) mm, rotated rx 0 ry 90 rz 0 deg; joints [-12.137, -27.556, 110.228, -16.192, -82.098, 51.266]
  Call Extruder(0.178)
  MoveL 6658 to (509.6, 509.6, 13.9) mm, rotated rx 0 ry 90 rz 0 deg; joints [-12.688, -27.528, 110.066, -16.754, -81.988, 51.374]
  Call Extruder(0.559)
  MoveL 6659 to (490.4, 509.6, 13.9) mm, rotated rx 0 ry 90 rz 0 deg; joints [-13.088, -27.89, 112.354, -17.086, -83.845, 50.852]
  MoveL 6660 to (490.4, 490.4, 13.9) mm, rotated rx 0 ry 90 rz 0 deg; joints [-11.303, -27.96, 112.844, -15.28, -84.202, 50.575]
  Call Extruder(0.154)
  MoveL 6661 to (495.71, 490.4, 13.9) mm, rotated rx 0 ry 90 rz 0 deg; joints [-11.205, -27.87, 112.215, -15.196, -83.679, 50.708]
  Call Extruder(0.010)
  MoveL 6662 to (496.06, 490.4, 13.9) mm, rotated rx 0 ry 90 rz 0 deg; joints [-11.198, -27.863, 112.173, -15.191, -83.645, 50.717]
  Call Extruder(0.007)
  MoveL 6663 to (496.06, 490.75, 13.9) mm, rotated rx 0 ry 90 rz 0 deg; joints [-11.231, -27.862, 112.165, -15.224, -83.639, 50.722]
  Call Extruder(0.035)
  MoveL 6664 to (496.06, 491.95, 13.9) mm, rotated rx 0 ry 90 rz 0 deg; joints [-11.342, -27.858, 112.137, -15.337, -83.619, 50.739]
  Call Extruder(0.010)
  MoveL 6665 to (496.06, 492.3, 13.9) mm, rotated rx 0 ry 90 rz 0 deg; joints [-11.374, -27.857, 112.128, -15.369, -83.613, 50.744]
  Call Extruder(0.007)
  MoveL 6666 to (496.41, 492.3, 13.9) mm, rotated rx 0 ry 90 rz 0 deg; joints [-11.368, -27.851, 112.087, -15.364, -83.578, 50.753]
  Call Extruder(0.061)
  MoveL 6667 to (498.51, 492.3, 13.9) mm, rotated rx 0 ry 90 rz 0 deg; joints [-11.329, -27.813, 111.836, -15.331, -83.372, 50.806]
  Call Extruder(0.055)
  MoveL 6668 to (498.52, 490.4, 13.9) mm, rotated rx 0 ry 90 rz 0 deg; joints [-11.153, -27.82, 111.881, -15.153, -83.404, 50.778]
  Call Extruder(0.064)
  MoveL 6669 to (500.72, 490.4, 13.9) mm, rotated rx 0 ry 90 rz 0 deg; joints [-11.113, -27.78, 111.617, -15.12, -83.187, 50.833]
  Call Extruder(0.055)
  MoveL 6670 to (500.72, 492.3, 13.9) mm, rotated rx 0 ry 90 rz 0 deg; joints [-11.288, -27.773, 111.572, -15.297, -83.155, 50.861]
  Call Extruder(0.061)
  MoveL 6671 to (502.81, 492.3, 13.9) mm, rotated rx 0 ry 90 rz 0 deg; joints [-11.25, -27.734, 111.323, -15.265, -82.951, 50.913]
  Call Extruder(0.007)
  MoveL 6672 to (503.15, 492.3, 13.9) mm, rotated rx 0 ry 90 rz 0 deg; joints [-11.244, -27.727, 111.281, -15.26, -82.917, 50.922]
  Set speed (120.0 mm/s)
  MoveL 6673 to (503.15, 491.95, 13.9) mm, rotated rx 0 ry 90 rz 0 deg; joints [-11.211, -27.729, 111.289, -15.228, -82.922, 50.916]
  Set speed (1000.0 mm/s)
  MoveL 6674 to (503.16, 491.9, 13.9) mm, rotated rx 0 ry 90 rz 0 deg; joints [-11.207, -27.729, 111.29, -15.223, -82.923, 50.915]
  Set speed (1000.0 mm/s)
  MoveL 6675 to (503.86, 491.9, 13.9) mm, rotated rx 0 ry 90 rz 0 deg; joints [-11.194, -27.716, 111.206, -15.212, -82.855, 50.933]
  Set speed (1000.0 mm/s)
  MoveL 6676 to (496.03, 492.33, 13.9) mm, rotated rx 0 ry 90 rz 0 deg; joints [-11.378, -27.857, 112.131, -15.372, -83.615, 50.744]
  Set speed (1000.0 mm/s)
  MoveL 6677 to (490.68, 490.68, 13.9) mm, rotated rx 0 ry 90 rz 0 deg; joints [-11.324, -27.955, 112.805, -15.302, -84.169, 50.586]
  Set speed (1000.0 mm/s)
  MoveL 6678 to (490.68, 490.68, 14) mm, rotated rx 0 ry 90 rz 0 deg; joints [-11.324, -27.965, 112.81, -15.302, -84.164, 50.587]
  Set speed (30.0 mm/s)
  Call Extruder(0.767)
  MoveL 6679 to (509.32, 509.32, 14) mm, rotated rx 0 ry 90 rz 0 deg; joints [-12.669, -27.546, 110.112, -16.733, -82.015, 51.363]
  MoveL 6680 to (509.44, 509.44, 14) mm, rotated rx 0 ry 90 rz 0 deg; joints [-12.677, -27.543, 110.094, -16.742, -82.001, 51.368]
  Set speed (120.0 mm/s)
  MoveL 6681 to (507.98, 504.67, 14) mm, rotated rx 0 ry 90 rz 0 deg; joints [-12.277, -27.594, 110.397, -16.328, -82.228, 51.247]
  Set speed (1000.0 mm/s)
  MoveL 6682 to (507.39, 502.51, 14) mm, rotated rx 0 ry 90 rz 0 deg; joints [-12.094, -27.615, 110.525, -16.139, -82.324, 51.194]
  Set speed (30.0 mm/s)
  Call Extruder(0.280)
  MoveL 6683 to (500.58, 509.32, 14) mm, rotated rx 0 ry 90 rz 0 deg; joints [-12.847, -27.718, 111.16, -16.879, -82.86, 51.129]
  Set speed (120.0 mm/s)
  MoveL 6684 to (499.42, 509.32, 14) mm, rotated rx 0 ry 90 rz 0 deg; joints [-12.872, -27.74, 111.298, -16.899, -82.972, 51.097]
  Set speed (30.0 mm/s)
  Call Extruder(0.360)
  MoveL 6685 to (490.68, 500.58, 14) mm, rotated rx 0 ry 90 rz 0 deg; joints [-12.247, -27.931, 112.566, -16.236, -83.986, 50.726]
  Set speed (120.0 mm/s)
  MoveL 6686 to (490.68, 499.42, 14) mm, rotated rx 0 ry 90 rz 0 deg; joints [-12.139, -27.935, 112.595, -16.127, -84.007, 50.709]
  Set speed (30.0 mm/s)
  Call Extruder(0.281)
  MoveL 6687 to (497.52, 492.58, 14) mm, rotated rx 0 ry 90 rz 0 deg; joints [-11.373, -27.84, 111.953, -15.373, -83.459, 50.786]
  MoveL 6688 to (497.64, 492.46, 14) mm, rotated rx 0 ry 90 rz 0 deg; joints [-11.36, -27.839, 111.941, -15.359, -83.449, 50.788]
  Set speed (120.0 mm/s)
  MoveL 6689 to (498.74, 491.36, 14) mm, rotated rx 0 ry 90 rz 0 deg; joints [-11.238, -27.823, 111.837, -15.24, -83.36, 50.799]
  Set speed (30.0 mm/s)
  Call Extruder(0.028)
  MoveL 6690 to (499.42, 490.68, 14) mm, rotated rx 0 ry 90 rz 0 deg; joints [-11.163, -27.813, 111.771, -15.166, -83.305, 50.806]
  Set speed (120.0 mm/s)
  MoveL 6691 to (500.76, 492.33, 14) mm, rotated rx 0 ry 90 rz 0 deg; joints [-11.29, -27.782, 111.572, -15.299, -83.146, 50.864]
  Set speed (1000.0 mm/s)
  MoveL 6692 to (502.48, 492.58, 14) mm, rotated rx 0 ry 90 rz 0 deg; joints [-11.282, -27.749, 111.36, -15.296, -82.973, 50.911]
  Set speed (30.0 mm/s)
  Call Extruder(0.202)
  MoveL 6693 to (507.39, 497.49, 14) mm, rotated rx 0 ry 90 rz 0 deg; joints [-11.639, -27.636, 110.651, -15.677, -82.41, 51.111]
  Set speed (120.0 mm/s)
  MoveL 6694 to (508.23, 498.33, 14) mm, rotated rx 0 ry 90 rz 0 deg; joints [-11.699, -27.616, 110.529, -15.741, -82.314, 51.146]
  Set speed (30.0 mm/s)
  Call Extruder(0.045)
  MoveL 6695 to (509.32, 499.42, 14) mm, rotated rx 0 ry 90 rz 0 deg; joints [-11.777, -27.589, 110.371, -15.825, -82.19, 51.192]
  Set speed (120.0 mm/s)
  MoveL 6696 to (509.32, 500.58, 14) mm, rotated rx 0 ry 90 rz 0 deg; joints [-11.882, -27.584, 110.341, -15.931, -82.17, 51.211]
  Set speed (30.0 mm/s)
  Call Extruder(0.007)
  MoveL 6697 to (509.15, 500.75, 14) mm, rotated rx 0 ry 90 rz 0 deg; joints [-11.9, -27.587, 110.357, -15.949, -82.183, 51.21]
  Set speed (120.0 mm/s)
  MoveL 6698 to (507.64, 498.08, 14) mm, rotated rx 0 ry 90 rz 0 deg; joints [-11.687, -27.628, 110.606, -15.727, -82.376, 51.127]
  Set speed (1000.0 mm/s)
  MoveL 6699 to (507.64, 495.51, 14) mm, rotated rx 0 ry 90 rz 0 deg; joints [-11.454, -27.639, 110.669, -15.49, -82.419, 51.085]
  Set speed (1000.0 mm/s)
  MoveL 6700 to (509.32, 490.68, 14) mm, rotated rx 0 ry 90 rz 0 deg; joints [-10.985, -27.625, 110.583, -15.02, -82.334, 51.049]
  Set speed (30.0 mm/s)
  Call Extruder(0.767)
  MoveL 6701 to (490.68, 509.32, 14) mm, rotated rx 0 ry 90 rz 0 deg; joints [-13.056, -27.897, 112.334, -17.055, -83.818, 50.857]
  MoveL 6702 to (490.56, 509.44, 14) mm, rotated rx 0 ry 90 rz 0 deg; joints [-13.07, -27.899, 112.345, -17.069, -83.827, 50.856]
  Set speed (120.0 mm/s)
  MoveL 6703 to (503.29, 492.37, 14) mm, rotated rx 0 ry 90 rz 0 deg; joints [-11.248, -27.735, 111.268, -15.265, -82.897, 50.927]
  Set speed (1000.0 mm/s)
  MoveL 6704 to (503.22, 492.3, 14) mm, rotated rx 0 ry 90 rz 0 deg; joints [-11.242, -27.737, 111.278, -15.259, -82.905, 50.925]
  Set speed (15.0 mm/s)
  Call Extruder(0.010)
  MoveL 6705 to (503.22, 491.95, 14) mm, rotated rx 0 ry 90 rz 0 deg; joints [-11.21, -27.738, 111.287, -15.227, -82.911, 50.919]
  Call Extruder(0.035)
  MoveL 6706 to (503.22, 490.75, 14) mm, rotated rx 0 ry 90 rz 0 deg; joints [-11.1, -27.742, 111.315, -15.115, -82.931, 50.901]
  Call Extruder(0.010)
  MoveL 6707 to (503.22, 490.4, 14) mm, rotated rx 0 ry 90 rz 0 deg; joints [-11.068, -27.744, 111.323, -15.083, -82.937, 50.896]
  Call Extruder(0.007)
  MoveL 6708 to (503.57, 490.4, 14) mm, rotated rx 0 ry 90 rz 0 deg; joints [-11.062, -27.737, 111.281, -15.077, -82.902, 50.904]
  Call Extruder(0.176)
  MoveL 6709 to (509.6, 490.4, 14) mm, rotated rx 0 ry 90 rz 0 deg; joints [-10.955, -27.62, 110.556, -14.99, -82.311, 51.051]
  Call Extruder(0.149)
  MoveL 6710 to (509.6, 495.54, 14) mm, rotated rx 0 ry 90 rz 0 deg; joints [-11.421, -27.6, 110.433, -15.463, -82.228, 51.134]
  Call Extruder(0.056)
  MoveL 6711 to (507.67, 495.54, 14) mm, rotated rx 0 ry 90 rz 0 deg; joints [-11.456, -27.638, 110.665, -15.492, -82.416, 51.086]
  Call Extruder(0.063)
  MoveL 6712 to (507.67, 497.7, 14) mm, rotated rx 0 ry 90 rz 0 deg; joints [-11.653, -27.629, 110.612, -15.692, -82.379, 51.122]
  Call Extruder(0.010)
  MoveL 6713 to (507.67, 498.05, 14) mm, rotated rx 0 ry 90 rz 0 deg; joints [-11.684, -27.628, 110.603, -15.724, -82.373, 51.128]
  Call Extruder(0.007)
  MoveL 6714 to (508.02, 498.05, 14) mm, rotated rx 0 ry 90 rz 0 deg; joints [-11.678, -27.621, 110.561, -15.719, -82.339, 51.136]
  Call Extruder(0.036)
  MoveL 6715 to (509.25, 498.05, 14) mm, rotated rx 0 ry 90 rz 0 deg; joints [-11.655, -27.596, 110.413, -15.7, -82.22, 51.167]
  Call Extruder(0.010)
  MoveL 6716 to (509.6, 498.05, 14) mm, rotated rx 0 ry 90 rz 0 deg; joints [-11.648, -27.589, 110.371, -15.695, -82.186, 51.176]
  Call Extruder(0.007)
  MoveL 6717 to (509.6, 498.4, 14) mm, rotated rx 0 ry 90 rz 0 deg; joints [-11.68, -27.588, 110.362, -15.727, -82.18, 51.182]
  Call Extruder(0.066)
  MoveL 6718 to (509.6, 500.68, 14) mm, rotated rx 0 ry 90 rz 0 deg; joints [-11.885, -27.578, 110.305, -15.936, -82.141, 51.22]
  Call Extruder(0.010)
  MoveL 6719 to (509.6, 501.03, 14) mm, rotated rx 0 ry 90 rz 0 deg; joints [-11.917, -27.577, 110.296, -15.968, -82.135, 51.226]
  Call Extruder(0.007)
  MoveL 6720 to (509.25, 501.03, 14) mm, rotated rx 0 ry 90 rz 0 deg; joints [-11.924, -27.584, 110.338, -15.974, -82.169, 51.217]
  Call Extruder(0.036)
  MoveL 6721 to (508.02, 501.02, 14) mm, rotated rx 0 ry 90 rz 0 deg; joints [-11.947, -27.609, 110.487, -15.992, -82.289, 51.186]
  Call Extruder(0.010)
  MoveL 6722 to (507.67, 501.02, 14) mm, rotated rx 0 ry 90 rz 0 deg; joints [-11.953, -27.616, 110.529, -15.998, -82.323, 51.177]
  Call Extruder(0.007)
  MoveL 6723 to (507.67, 501.37, 14) mm, rotated rx 0 ry 90 rz 0 deg; joints [-11.985, -27.614, 110.52, -16.03, -82.316, 51.183]
  Call Extruder(0.063)
  MoveL 6724 to (507.67, 503.52, 14) mm, rotated rx 0 ry 90 rz 0 deg; joints [-12.179, -27.605, 110.465, -16.228, -82.279, 51.219]
  Call Extruder(0.056)
  MoveL 6725 to (509.6, 503.53, 14) mm, rotated rx 0 ry 90 rz 0 deg; joints [-12.142, -27.566, 110.232, -16.198, -82.092, 51.269]
  Call Extruder(0.177)
  MoveL 6726 to (509.6, 509.6, 14) mm, rotated rx 0 ry 90 rz 0 deg; joints [-12.688, -27.539, 110.071, -16.754, -81.983, 51.375]
  Call Extruder(0.559)
  MoveL 6727 to (490.4, 509.6, 14) mm, rotated rx 0 ry 90 rz 0 deg; joints [-13.088, -27.901, 112.359, -17.087, -83.839, 50.854]
  MoveL 6728 to (490.4, 490.4, 14) mm, rotated rx 0 ry 90 rz 0 deg; joints [-11.303, -27.971, 112.85, -15.281, -84.197, 50.576]
  Call Extruder(0.153)
  MoveL 6729 to (495.65, 490.4, 14) mm, rotated rx 0 ry 90 rz 0 deg; joints [-11.206, -27.881, 112.227, -15.197, -83.68, 50.708]
  Call Extruder(0.010)
  MoveL 6730 to (496, 490.4, 14) mm, rotated rx 0 ry 90 rz 0 deg; joints [-11.199, -27.875, 112.185, -15.192, -83.645, 50.717]
  Call Extruder(0.007)
  MoveL 6731 to (496, 490.75, 14) mm, rotated rx 0 ry 90 rz 0 deg; joints [-11.232, -27.874, 112.177, -15.225, -83.639, 50.722]
  Call Extruder(0.035)
  MoveL 6732 to (496, 491.95, 14) mm, rotated rx 0 ry 90 rz 0 deg; joints [-11.343, -27.87, 112.148, -15.338, -83.619, 50.739]
  Call Extruder(0.010)
  MoveL 6733 to (496, 492.3, 14) mm, rotated rx 0 ry 90 rz 0 deg; joints [-11.375, -27.868, 112.14, -15.37, -83.613, 50.744]
  Call Extruder(0.007)
  MoveL 6734 to (496.35, 492.3, 14) mm, rotated rx 0 ry 90 rz 0 deg; joints [-11.369, -27.862, 112.098, -15.365, -83.579, 50.753]
  Call Extruder(0.061)
  MoveL 6735 to (498.46, 492.3, 14) mm, rotated rx 0 ry 90 rz 0 deg; joints [-11.33, -27.825, 111.848, -15.332, -83.372, 50.806]
  Call Extruder(0.055)
  MoveL 6736 to (498.46, 490.4, 14) mm, rotated rx 0 ry 90 rz 0 deg; joints [-11.154, -27.831, 111.892, -15.154, -83.404, 50.778]
  Call Extruder(0.068)
  MoveL 6737 to (500.79, 490.4, 14) mm, rotated rx 0 ry 90 rz 0 deg; joints [-11.112, -27.789, 111.615, -15.119, -83.175, 50.836]
  Call Extruder(0.055)
  MoveL 6738 to (500.79, 492.3, 14) mm, rotated rx 0 ry 90 rz 0 deg; joints [-11.287, -27.782, 111.569, -15.296, -83.143, 50.864]
  Call Extruder(0.061)
  MoveL 6739 to (502.87, 492.3, 14) mm, rotated rx 0 ry 90 rz 0 deg; joints [-11.249, -27.743, 111.32, -15.265, -82.939, 50.916]
  Call Extruder(0.007)
  MoveL 6740 to (503.22, 492.3, 14) mm, rotated rx 0 ry 90 rz 0 deg; joints [-11.242, -27.737, 111.278, -15.259, -82.905, 50.925]
  Set speed (120.0 mm/s)
  MoveL 6741 to (503.22, 491.95, 14) mm, rotated rx 0 ry 90 rz 0 deg; joints [-11.21, -27.738, 111.287, -15.227, -82.911, 50.919]
  Set speed (1000.0 mm/s)
  MoveL 6742 to (503.22, 491.9, 14) mm, rotated rx 0 ry 90 rz 0 deg; joints [-11.206, -27.738, 111.288, -15.222, -82.912, 50.918]
  Set speed (1000.0 mm/s)
  MoveL 6743 to (503.92, 491.9, 14) mm, rotated rx 0 ry 90 rz 0 deg; joints [-11.193, -27.725, 111.204, -15.212, -82.843, 50.936]
  Set speed (1000.0 mm/s)
  MoveL 6744 to (495.97, 492.33, 14) mm, rotated rx 0 ry 90 rz 0 deg; joints [-11.379, -27.869, 112.143, -15.374, -83.615, 50.744]
  Set speed (1000.0 mm/s)
  MoveL 6745 to (490.68, 490.68, 14) mm, rotated rx 0 ry 90 rz 0 deg; joints [-11.324, -27.965, 112.81, -15.302, -84.164, 50.587]
  Set speed (1000.0 mm/s)
  MoveL 6746 to (490.68, 490.68, 14.1) mm, rotated rx 0 ry 90 rz 0 deg; joints [-11.324, -27.976, 112.815, -15.303, -84.159, 50.588]
  Set speed (30.0 mm/s)
  Call Extruder(0.767)
  MoveL 6747 to (509.32, 509.32, 14.1) mm, rotated rx 0 ry 90 rz 0 deg; joints [-12.669, -27.556, 110.117, -16.733, -82.01, 51.364]
  MoveL 6748 to (509.44, 509.44, 14.1) mm, rotated rx 0 ry 90 rz 0 deg; joints [-12.677, -27.553, 110.099, -16.742, -81.996, 51.37]
  Set speed (120.0 mm/s)
  MoveL 6749 to (507.82, 504.19, 14.1) mm, rotated rx 0 ry 90 rz 0 deg; joints [-12.237, -27.61, 110.434, -16.287, -82.247, 51.236]
  Set speed (1000.0 mm/s)
  MoveL 6750 to (507.39, 502.51, 14.1) mm, rotated rx 0 ry 90 rz 0 deg; joints [-12.094, -27.625, 110.53, -16.139, -82.319, 51.196]
  Set speed (30.0 mm/s)
  Call Extruder(0.280)
  MoveL 6751 to (500.58, 509.32, 14.1) mm, rotated rx 0 ry 90 rz 0 deg; joints [-12.847, -27.728, 111.165, -16.879, -82.855, 51.13]
  Set speed (120.0 mm/s)
  MoveL 6752 to (499.42, 509.32, 14.1) mm, rotated rx 0 ry 90 rz 0 deg; joints [-12.872, -27.75, 111.303, -16.9, -82.967, 51.099]
  Set speed (30.0 mm/s)
  Call Extruder(0.360)
  MoveL 6753 to (490.68, 500.58, 14.1) mm, rotated rx 0 ry 90 rz 0 deg; joints [-12.247, -27.941, 112.571, -16.236, -83.98, 50.728]
  Set speed (120.0 mm/s)
  MoveL 6754 to (490.68, 499.42, 14.1) mm, rotated rx 0 ry 90 rz 0 deg; joints [-12.139, -27.946, 112.601, -16.127, -84.002, 50.711]
  Set speed (30.0 mm/s)
  Call Extruder(0.281)
  MoveL 6755 to (497.52, 492.58, 14.1) mm, rotated rx 0 ry 90 rz 0 deg; joints [-11.373, -27.851, 111.958, -15.373, -83.454, 50.788]
  MoveL 6756 to (497.64, 492.46, 14.1) mm, rotated rx 0 ry 90 rz 0 deg; joints [-11.36, -27.849, 111.946, -15.36, -83.444, 50.789]
  Set speed (120.0 mm/s)
  MoveL 6757 to (498.68, 491.42, 14.1) mm, rotated rx 0 ry 90 rz 0 deg; joints [-11.244, -27.834, 111.847, -15.246, -83.36, 50.8]
  Set speed (30.0 mm/s)
  Call Extruder(0.030)
  MoveL 6758 to (499.42, 490.68, 14.1) mm, rotated rx 0 ry 90 rz 0 deg; joints [-11.163, -27.824, 111.776, -15.166, -83.3, 50.807]
  Set speed (120.0 mm/s)
  MoveL 6759 to (500.82, 492.33, 14.1) mm, rotated rx 0 ry 90 rz 0 deg; joints [-11.289, -27.792, 111.57, -15.298, -83.134, 50.867]
  Set speed (1000.0 mm/s)
  MoveL 6760 to (502.48, 492.58, 14.1) mm, rotated rx 0 ry 90 rz 0 deg; joints [-11.282, -27.76, 111.365, -15.297, -82.968, 50.912]
  Set speed (30.0 mm/s)
  Call Extruder(0.202)
  MoveL 6761 to (507.39, 497.49, 14.1) mm, rotated rx 0 ry 90 rz 0 deg; joints [-11.639, -27.646, 110.656, -15.677, -82.405, 51.113]
  Set speed (120.0 mm/s)
  MoveL 6762 to (508.17, 498.27, 14.1) mm, rotated rx 0 ry 90 rz 0 deg; joints [-11.695, -27.628, 110.543, -15.737, -82.316, 51.145]
  Set speed (30.0 mm/s)
  Call Extruder(0.047)
  MoveL 6763 to (509.32, 499.42, 14.1) mm, rotated rx 0 ry 90 rz 0 deg; joints [-11.777, -27.6, 110.376, -15.825, -82.185, 51.193]
  Set speed (120.0 mm/s)
  MoveL 6764 to (509.32, 500.58, 14.1) mm, rotated rx 0 ry 90 rz 0 deg; joints [-11.882, -27.595, 110.347, -15.932, -82.165, 51.213]
  Set speed (30.0 mm/s)
  Call Extruder(0.009)
  MoveL 6765 to (509.1, 500.8, 14.1) mm, rotated rx 0 ry 90 rz 0 deg; joints [-11.906, -27.598, 110.368, -15.956, -82.183, 51.211]
  Set speed (120.0 mm/s)
  MoveL 6766 to (507.64, 498.02, 14.1) mm, rotated rx 0 ry 90 rz 0 deg; joints [-11.682, -27.639, 110.612, -15.722, -82.371, 51.128]
  Set speed (1000.0 mm/s)
  MoveL 6767 to (507.64, 495.45, 14.1) mm, rotated rx 0 ry 90 rz 0 deg; joints [-11.449, -27.649, 110.676, -15.485, -82.415, 51.086]
  Set speed (1000.0 mm/s)
  MoveL 6768 to (509.32, 490.68, 14.1) mm, rotated rx 0 ry 90 rz 0 deg; joints [-10.985, -27.635, 110.588, -15.02, -82.329, 51.05]
  Set speed (30.0 mm/s)
  Call Extruder(0.767)
  MoveL 6769 to (490.68, 509.32, 14.1) mm, rotated rx 0 ry 90 rz 0 deg; joints [-13.056, -27.908, 112.339, -17.055, -83.813, 50.859]
  MoveL 6770 to (490.56, 509.44, 14.1) mm, rotated rx 0 ry 90 rz 0 deg; joints [-13.07, -27.909, 112.35, -17.069, -83.822, 50.858]
  Set speed (120.0 mm/s)
  MoveL 6771 to (503.35, 492.37, 14.1) mm, rotated rx 0 ry 90 rz 0 deg; joints [-11.246, -27.744, 111.266, -15.264, -82.886, 50.93]
  Set speed (1000.0 mm/s)
  MoveL 6772 to (503.28, 492.3, 14.1) mm, rotated rx 0 ry 90 rz 0 deg; joints [-11.241, -27.746, 111.276, -15.259, -82.894, 50.928]
  Set speed (15.0 mm/s)
  Call Extruder(0.010)
  MoveL 6773 to (503.28, 491.95, 14.1) mm, rotated rx 0 ry 90 rz 0 deg; joints [-11.209, -27.747, 111.284, -15.226, -82.899, 50.922]
  Call Extruder(0.035)
  MoveL 6774 to (503.28, 490.75, 14.1) mm, rotated rx 0 ry 90 rz 0 deg; joints [-11.099, -27.752, 111.313, -15.114, -82.919, 50.904]
  Call Extruder(0.010)
  MoveL 6775 to (503.28, 490.4, 14.1) mm, rotated rx 0 ry 90 rz 0 deg; joints [-11.067, -27.753, 111.321, -15.082, -82.925, 50.899]
  Call Extruder(0.007)
  MoveL 6776 to (503.63, 490.4, 14.1) mm, rotated rx 0 ry 90 rz 0 deg; joints [-11.061, -27.746, 111.279, -15.077, -82.891, 50.907]
  Call Extruder(0.174)
  MoveL 6777 to (509.6, 490.4, 14.1) mm, rotated rx 0 ry 90 rz 0 deg; joints [-10.955, -27.631, 110.561, -14.99, -82.306, 51.053]
  Call Extruder(0.148)
  MoveL 6778 to (509.6, 495.48, 14.1) mm, rotated rx 0 ry 90 rz 0 deg; joints [-11.415, -27.61, 110.44, -15.458, -82.223, 51.135]
  Call Extruder(0.056)
  MoveL 6779 to (507.67, 495.48, 14.1) mm, rotated rx 0 ry 90 rz 0 deg; joints [-11.451, -27.649, 110.672, -15.487, -82.412, 51.087]
  Call Extruder(0.073)
  MoveL 6780 to (507.67, 497.99, 14.1) mm, rotated rx 0 ry 90 rz 0 deg; joints [-11.679, -27.639, 110.61, -15.719, -82.369, 51.128]
  Call Extruder(0.056)
  MoveL 6781 to (509.6, 497.99, 14.1) mm, rotated rx 0 ry 90 rz 0 deg; joints [-11.643, -27.6, 110.378, -15.69, -82.181, 51.177]
  Call Extruder(0.080)
  MoveL 6782 to (509.6, 500.73, 14.1) mm, rotated rx 0 ry 90 rz 0 deg; joints [-11.89, -27.589, 110.309, -15.941, -82.135, 51.223]
  Call Extruder(0.010)
  MoveL 6783 to (509.6, 501.08, 14.1) mm, rotated rx 0 ry 90 rz 0 deg; joints [-11.922, -27.587, 110.3, -15.974, -82.129, 51.229]
  Call Extruder(0.007)
  MoveL 6784 to (509.25, 501.08, 14.1) mm, rotated rx 0 ry 90 rz 0 deg; joints [-11.929, -27.594, 110.342, -15.979, -82.163, 51.22]
  Call Extruder(0.036)
  MoveL 6785 to (508.02, 501.08, 14.1) mm, rotated rx 0 ry 90 rz 0 deg; joints [-11.952, -27.619, 110.49, -15.998, -82.282, 51.188]
  Call Extruder(0.010)
  MoveL 6786 to (507.67, 501.08, 14.1) mm, rotated rx 0 ry 90 rz 0 deg; joints [-11.959, -27.626, 110.533, -16.003, -82.316, 51.179]
  Call Extruder(0.007)
  MoveL 6787 to (507.67, 501.43, 14.1) mm, rotated rx 0 ry 90 rz 0 deg; joints [-11.99, -27.624, 110.524, -16.035, -82.31, 51.185]
  Call Extruder(0.063)
  MoveL 6788 to (507.67, 503.58, 14.1) mm, rotated rx 0 ry 90 rz 0 deg; joints [-12.185, -27.615, 110.468, -16.233, -82.273, 51.221]
  Call Extruder(0.056)
  MoveL 6789 to (509.6, 503.58, 14.1) mm, rotated rx 0 ry 90 rz 0 deg; joints [-12.147, -27.576, 110.236, -16.203, -82.085, 51.271]
  Call Extruder(0.175)
  MoveL 6790 to (509.6, 509.6, 14.1) mm, rotated rx 0 ry 90 rz 0 deg; joints [-12.688, -27.549, 110.076, -16.754, -81.978, 51.377]
  Call Extruder(0.559)
  MoveL 6791 to (490.4, 509.6, 14.1) mm, rotated rx 0 ry 90 rz 0 deg; joints [-13.088, -27.911, 112.364, -17.087, -83.834, 50.856]
  MoveL 6792 to (490.4, 490.4, 14.1) mm, rotated rx 0 ry 90 rz 0 deg; joints [-11.303, -27.982, 112.855, -15.281, -84.191, 50.578]
  Call Extruder(0.151)
  MoveL 6793 to (495.6, 490.4, 14.1) mm, rotated rx 0 ry 90 rz 0 deg; joints [-11.207, -27.893, 112.239, -15.199, -83.68, 50.708]
  Call Extruder(0.010)
  MoveL 6794 to (495.95, 490.4, 14.1) mm, rotated rx 0 ry 90 rz 0 deg; joints [-11.2, -27.887, 112.197, -15.193, -83.646, 50.717]
  Call Extruder(0.007)
  MoveL 6795 to (495.95, 490.75, 14.1) mm, rotated rx 0 ry 90 rz 0 deg; joints [-11.233, -27.885, 112.189, -15.226, -83.64, 50.722]
  Call Extruder(0.035)
  MoveL 6796 to (495.95, 491.95, 14.1) mm, rotated rx 0 ry 90 rz 0 deg; joints [-11.344, -27.881, 112.16, -15.339, -83.619, 50.739]
  Call Extruder(0.010)
  MoveL 6797 to (495.94, 492.3, 14.1) mm, rotated rx 0 ry 90 rz 0 deg; joints [-11.377, -27.88, 112.152, -15.371, -83.613, 50.744]
  Call Extruder(0.007)
  MoveL 6798 to (496.3, 492.3, 14.1) mm, rotated rx 0 ry 90 rz 0 deg; joints [-11.37, -27.874, 112.11, -15.366, -83.579, 50.753]
  Call Extruder(0.061)
  MoveL 6799 to (498.4, 492.3, 14.1) mm, rotated rx 0 ry 90 rz 0 deg; joints [-11.331, -27.836, 111.859, -15.333, -83.372, 50.806]
  Call Extruder(0.055)
  MoveL 6800 to (498.4, 490.4, 14.1) mm, rotated rx 0 ry 90 rz 0 deg; joints [-11.155, -27.843, 111.904, -15.155, -83.404, 50.778]
  Call Extruder(0.071)
  MoveL 6801 to (500.85, 490.4, 14.1) mm, rotated rx 0 ry 90 rz 0 deg; joints [-11.111, -27.798, 111.612, -15.118, -83.164, 50.839]
  Call Extruder(0.055)
  MoveL 6802 to (500.85, 492.3, 14.1) mm, rotated rx 0 ry 90 rz 0 deg; joints [-11.286, -27.791, 111.567, -15.295, -83.132, 50.867]
  Call Extruder(0.061)
  MoveL 6803 to (502.93, 492.3, 14.1) mm, rotated rx 0 ry 90 rz 0 deg; joints [-11.248, -27.753, 111.318, -15.264, -82.928, 50.919]
  Call Extruder(0.007)
  MoveL 6804 to (503.28, 492.3, 14.1) mm, rotated rx 0 ry 90 rz 0 deg; joints [-11.241, -27.746, 111.276, -15.259, -82.894, 50.928]
  Set speed (120.0 mm/s)
  MoveL 6805 to (503.28, 491.95, 14.1) mm, rotated rx 0 ry 90 rz 0 deg; joints [-11.209, -27.747, 111.284, -15.226, -82.899, 50.922]
  Set speed (1000.0 mm/s)
  MoveL 6806 to (503.28, 491.9, 14.1) mm, rotated rx 0 ry 90 rz 0 deg; joints [-11.205, -27.747, 111.285, -15.221, -82.9, 50.921]
  Set speed (1000.0 mm/s)
  MoveL 6807 to (503.98, 491.9, 14.1) mm, rotated rx 0 ry 90 rz 0 deg; joints [-11.192, -27.734, 111.201, -15.211, -82.832, 50.939]
  Set speed (1000.0 mm/s)
  MoveL 6808 to (495.92, 492.33, 14.1) mm, rotated rx 0 ry 90 rz 0 deg; joints [-11.38, -27.88, 112.155, -15.375, -83.615, 50.744]
  Set speed (1000.0 mm/s)
  MoveL 6809 to (490.68, 490.68, 14.1) mm, rotated rx 0 ry 90 rz 0 deg; joints [-11.324, -27.976, 112.815, -15.303, -84.159, 50.588]
  Set speed (1000.0 mm/s)
  MoveL 6810 to (490.68, 490.68, 14.2) mm, rotated rx 0 ry 90 rz 0 deg; joints [-11.324, -27.987, 112.82, -15.303, -84.154, 50.59]
  Set speed (30.0 mm/s)
  Call Extruder(0.767)
  MoveL 6811 to (509.32, 509.32, 14.2) mm, rotated rx 0 ry 90 rz 0 deg; joints [-12.669, -27.567, 110.123, -16.733, -82.005, 51.366]
  MoveL 6812 to (509.44, 509.44, 14.2) mm, rotated rx 0 ry 90 rz 0 deg; joints [-12.677, -27.564, 110.104, -16.742, -81.991, 51.371]
  Set speed (120.0 mm/s)
  MoveL 6813 to (507.64, 503.66, 14.2) mm, rotated rx 0 ry 90 rz 0 deg; joints [-12.193, -27.626, 110.475, -16.242, -82.269, 51.224]
  Set speed (1000.0 mm/s)
  MoveL 6814 to (507.39, 502.51, 14.2) mm, rotated rx 0 ry 90 rz 0 deg; joints [-12.093, -27.636, 110.535, -16.139, -82.314, 51.197]
  Set speed (30.0 mm/s)
  Call Extruder(0.280)
  MoveL 6815 to (500.58, 509.32, 14.2) mm, rotated rx 0 ry 90 rz 0 deg; joints [-12.847, -27.739, 111.17, -16.88, -82.849, 51.132]
  Set speed (120.0 mm/s)
  MoveL 6816 to (499.42, 509.32, 14.2) mm, rotated rx 0 ry 90 rz 0 deg; joints [-12.872, -27.761, 111.308, -16.9, -82.961, 51.1]
  Set speed (30.0 mm/s)
  Call Extruder(0.360)
  MoveL 6817 to (490.68, 500.58, 14.2) mm, rotated rx 0 ry 90 rz 0 deg; joints [-12.247, -27.952, 112.576, -16.236, -83.975, 50.729]
  Set speed (120.0 mm/s)
  MoveL 6818 to (490.68, 499.42, 14.2) mm, rotated rx 0 ry 90 rz 0 deg; joints [-12.139, -27.956, 112.606, -16.127, -83.997, 50.712]
  Set speed (30.0 mm/s)
  Call Extruder(0.281)
  MoveL 6819 to (497.52, 492.58, 14.2) mm, rotated rx 0 ry 90 rz 0 deg; joints [-11.373, -27.862, 111.963, -15.373, -83.449, 50.789]
  MoveL 6820 to (497.64, 492.46, 14.2) mm, rotated rx 0 ry 90 rz 0 deg; joints [-11.359, -27.86, 111.951, -15.36, -83.439, 50.791]
  Set speed (120.0 mm/s)
  MoveL 6821 to (498.62, 491.48, 14.2) mm, rotated rx 0 ry 90 rz 0 deg; joints [-11.251, -27.846, 111.858, -15.253, -83.359, 50.801]
  Set speed (30.0 mm/s)
  Call Extruder(0.033)
  MoveL 6822 to (499.42, 490.68, 14.2) mm, rotated rx 0 ry 90 rz 0 deg; joints [-11.163, -27.834, 111.782, -15.166, -83.294, 50.809]
  Set speed (120.0 mm/s)
  MoveL 6823 to (500.89, 492.33, 14.2) mm, rotated rx 0 ry 90 rz 0 deg; joints [-11.288, -27.801, 111.567, -15.298, -83.123, 50.87]
  Set speed (1000.0 mm/s)
  MoveL 6824 to (502.48, 492.58, 14.2) mm, rotated rx 0 ry 90 rz 0 deg; joints [-11.282, -27.771, 111.371, -15.297, -82.963, 50.913]
  Set speed (30.0 mm/s)
  Call Extruder(0.202)
  MoveL 6825 to (507.39, 497.49, 14.2) mm, rotated rx 0 ry 90 rz 0 deg; joints [-11.639, -27.657, 110.661, -15.677, -82.4, 51.114]
  Set speed (120.0 mm/s)
  MoveL 6826 to (508.11, 498.22, 14.2) mm, rotated rx 0 ry 90 rz 0 deg; joints [-11.691, -27.639, 110.556, -15.733, -82.317, 51.144]
  Set speed (30.0 mm/s)
  Call Extruder(0.050)
  MoveL 6827 to (509.32, 499.42, 14.2) mm, rotated rx 0 ry 90 rz 0 deg; joints [-11.777, -27.61, 110.381, -15.825, -82.179, 51.195]
  Set speed (120.0 mm/s)
  MoveL 6828 to (509.32, 500.58, 14.2) mm, rotated rx 0 ry 90 rz 0 deg; joints [-11.882, -27.605, 110.352, -15.932, -82.16, 51.214]
  Set speed (30.0 mm/s)
  Call Extruder(0.011)
  MoveL 6829 to (509.04, 500.86, 14.2) mm, rotated rx 0 ry 90 rz 0 deg; joints [-11.912, -27.61, 110.378, -15.962, -82.182, 51.212]
  Set speed (120.0 mm/s)
  MoveL 6830 to (507.64, 497.96, 14.2) mm, rotated rx 0 ry 90 rz 0 deg; joints [-11.677, -27.65, 110.619, -15.717, -82.367, 51.128]
  Set speed (1000.0 mm/s)
  MoveL 6831 to (507.64, 495.39, 14.2) mm, rotated rx 0 ry 90 rz 0 deg; joints [-11.443, -27.66, 110.682, -15.479, -82.411, 51.086]
  Set speed (1000.0 mm/s)
  MoveL 6832 to (509.32, 490.68, 14.2) mm, rotated rx 0 ry 90 rz 0 deg; joints [-10.985, -27.646, 110.593, -15.02, -82.324, 51.052]
  Set speed (30.0 mm/s)
  Call Extruder(0.767)
  MoveL 6833 to (490.68, 509.32, 14.2) mm, rotated rx 0 ry 90 rz 0 deg; joints [-13.056, -27.918, 112.344, -17.056, -83.807, 50.861]
  MoveL 6834 to (490.56, 509.44, 14.2) mm, rotated rx 0 ry 90 rz 0 deg; joints [-13.07, -27.92, 112.356, -17.069, -83.817, 50.859]
  Set speed (120.0 mm/s)
  MoveL 6835 to (503.42, 492.37, 14.2) mm, rotated rx 0 ry 90 rz 0 deg; joints [-11.245, -27.754, 111.263, -15.263, -82.874, 50.933]
  Set speed (1000.0 mm/s)
  MoveL 6836 to (503.35, 492.3, 14.2) mm, rotated rx 0 ry 90 rz 0 deg; joints [-11.24, -27.755, 111.273, -15.258, -82.882, 50.931]
  Set speed (15.0 mm/s)
  Call Extruder(0.010)
  MoveL 6837 to (503.35, 491.95, 14.2) mm, rotated rx 0 ry 90 rz 0 deg; joints [-11.208, -27.757, 111.282, -15.225, -82.888, 50.925]
  Call Extruder(0.035)
  MoveL 6838 to (503.35, 490.75, 14.2) mm, rotated rx 0 ry 90 rz 0 deg; joints [-11.098, -27.761, 111.31, -15.114, -82.908, 50.907]
  Call Extruder(0.010)
  MoveL 6839 to (503.35, 490.4, 14.2) mm, rotated rx 0 ry 90 rz 0 deg; joints [-11.066, -27.762, 111.318, -15.081, -82.914, 50.902]
  Call Extruder(0.007)
  MoveL 6840 to (503.7, 490.4, 14.2) mm, rotated rx 0 ry 90 rz 0 deg; joints [-11.06, -27.756, 111.276, -15.076, -82.879, 50.91]
  Call Extruder(0.172)
  MoveL 6841 to (509.6, 490.4, 14.2) mm, rotated rx 0 ry 90 rz 0 deg; joints [-10.955, -27.641, 110.566, -14.99, -82.301, 51.054]
  Call Extruder(0.146)
  MoveL 6842 to (509.6, 495.42, 14.2) mm, rotated rx 0 ry 90 rz 0 deg; joints [-11.41, -27.621, 110.446, -15.453, -82.219, 51.135]
  Call Extruder(0.056)
  MoveL 6843 to (507.67, 495.42, 14.2) mm, rotated rx 0 ry 90 rz 0 deg; joints [-11.445, -27.66, 110.678, -15.482, -82.407, 51.087]
  Call Extruder(0.063)
  MoveL 6844 to (507.67, 497.59, 14.2) mm, rotated rx 0 ry 90 rz 0 deg; joints [-11.642, -27.651, 110.625, -15.681, -82.371, 51.123]
  Call Extruder(0.010)
  MoveL 6845 to (507.67, 497.94, 14.2) mm, rotated rx 0 ry 90 rz 0 deg; joints [-11.674, -27.649, 110.616, -15.714, -82.365, 51.129]
  Call Extruder(0.007)
  MoveL 6846 to (508.02, 497.94, 14.2) mm, rotated rx 0 ry 90 rz 0 deg; joints [-11.667, -27.642, 110.574, -15.708, -82.331, 51.137]
  Call Extruder(0.036)
  MoveL 6847 to (509.25, 497.93, 14.2) mm, rotated rx 0 ry 90 rz 0 deg; joints [-11.644, -27.618, 110.426, -15.69, -82.211, 51.168]
  Call Extruder(0.010)
  MoveL 6848 to (509.6, 497.93, 14.2) mm, rotated rx 0 ry 90 rz 0 deg; joints [-11.638, -27.611, 110.384, -15.684, -82.177, 51.177]
  Call Extruder(0.007)
  MoveL 6849 to (509.6, 498.28, 14.2) mm, rotated rx 0 ry 90 rz 0 deg; joints [-11.669, -27.609, 110.375, -15.717, -82.171, 51.183]
  Call Extruder(0.073)
  MoveL 6850 to (509.6, 500.79, 14.2) mm, rotated rx 0 ry 90 rz 0 deg; joints [-11.895, -27.599, 110.312, -15.947, -82.129, 51.225]
  Call Extruder(0.010)
  MoveL 6851 to (509.6, 501.14, 14.2) mm, rotated rx 0 ry 90 rz 0 deg; joints [-11.927, -27.597, 110.304, -15.979, -82.123, 51.231]
  Call Extruder(0.007)
  MoveL 6852 to (509.25, 501.14, 14.2) mm, rotated rx 0 ry 90 rz 0 deg; joints [-11.934, -27.604, 110.346, -15.984, -82.157, 51.222]
  Call Extruder(0.036)
  MoveL 6853 to (508.02, 501.14, 14.2) mm, rotated rx 0 ry 90 rz 0 deg; joints [-11.957, -27.629, 110.494, -16.003, -82.276, 51.191]
  Call Extruder(0.010)
  MoveL 6854 to (507.67, 501.14, 14.2) mm, rotated rx 0 ry 90 rz 0 deg; joints [-11.964, -27.636, 110.536, -16.009, -82.31, 51.182]
  Call Extruder(0.007)
  MoveL 6855 to (507.67, 501.49, 14.2) mm, rotated rx 0 ry 90 rz 0 deg; joints [-11.995, -27.635, 110.527, -16.041, -82.304, 51.188]
  Call Extruder(0.063)
  MoveL 6856 to (507.67, 503.64, 14.2) mm, rotated rx 0 ry 90 rz 0 deg; joints [-12.19, -27.625, 110.472, -16.238, -82.267, 51.224]
  Call Extruder(0.056)
  MoveL 6857 to (509.6, 503.64, 14.2) mm, rotated rx 0 ry 90 rz 0 deg; joints [-12.152, -27.587, 110.239, -16.208, -82.079, 51.274]
  Call Extruder(0.173)
  MoveL 6858 to (509.6, 509.6, 14.2) mm, rotated rx 0 ry 90 rz 0 deg; joints [-12.688, -27.56, 110.081, -16.754, -81.973, 51.378]
  Call Extruder(0.559)
  MoveL 6859 to (490.4, 509.6, 14.2) mm, rotated rx 0 ry 90 rz 0 deg; joints [-13.088, -27.922, 112.37, -17.087, -83.829, 50.857]
  MoveL 6860 to (490.4, 490.4, 14.2) mm, rotated rx 0 ry 90 rz 0 deg; joints [-11.303, -27.992, 112.86, -15.281, -84.186, 50.579]
  Call Extruder(0.150)
  MoveL 6861 to (495.54, 490.4, 14.2) mm, rotated rx 0 ry 90 rz 0 deg; joints [-11.208, -27.904, 112.25, -15.2, -83.68, 50.708]
  Call Extruder(0.010)
  MoveL 6862 to (495.89, 490.4, 14.2) mm, rotated rx 0 ry 90 rz 0 deg; joints [-11.201, -27.898, 112.209, -15.194, -83.646, 50.717]
  Call Extruder(0.007)
  MoveL 6863 to (495.89, 490.75, 14.2) mm, rotated rx 0 ry 90 rz 0 deg; joints [-11.234, -27.897, 112.201, -15.227, -83.64, 50.722]
  Call Extruder(0.035)
  MoveL 6864 to (495.89, 491.95, 14.2) mm, rotated rx 0 ry 90 rz 0 deg; joints [-11.345, -27.893, 112.172, -15.34, -83.619, 50.739]
  Call Extruder(0.010)
  MoveL 6865 to (495.89, 492.3, 14.2) mm, rotated rx 0 ry 90 rz 0 deg; joints [-11.378, -27.892, 112.164, -15.373, -83.613, 50.744]
  Call Extruder(0.007)
  MoveL 6866 to (496.24, 492.3, 14.2) mm, rotated rx 0 ry 90 rz 0 deg; joints [-11.371, -27.885, 112.122, -15.367, -83.579, 50.753]
  Call Extruder(0.061)
  MoveL 6867 to (498.34, 492.3, 14.2) mm, rotated rx 0 ry 90 rz 0 deg; joints [-11.332, -27.848, 111.871, -15.334, -83.372, 50.806]
  Call Extruder(0.055)
  MoveL 6868 to (498.35, 490.4, 14.2) mm, rotated rx 0 ry 90 rz 0 deg; joints [-11.156, -27.855, 111.916, -15.156, -83.404, 50.778]
  Call Extruder(0.075)
  MoveL 6869 to (500.91, 490.4, 14.2) mm, rotated rx 0 ry 90 rz 0 deg; joints [-11.11, -27.808, 111.61, -15.117, -83.153, 50.842]
  Call Extruder(0.055)
  MoveL 6870 to (500.91, 492.3, 14.2) mm, rotated rx 0 ry 90 rz 0 deg; joints [-11.285, -27.801, 111.565, -15.295, -83.121, 50.87]
  Call Extruder(0.061)
  MoveL 6871 to (503, 492.3, 14.2) mm, rotated rx 0 ry 90 rz 0 deg; joints [-11.246, -27.762, 111.315, -15.263, -82.916, 50.922]
  Call Extruder(0.007)
  MoveL 6872 to (503.35, 492.3, 14.2) mm, rotated rx 0 ry 90 rz 0 deg; joints [-11.24, -27.755, 111.273, -15.258, -82.882, 50.931]
  Set speed (120.0 mm/s)
  MoveL 6873 to (503.35, 491.95, 14.2) mm, rotated rx 0 ry 90 rz 0 deg; joints [-11.208, -27.757, 111.282, -15.225, -82.888, 50.925]
  Set speed (1000.0 mm/s)
  MoveL 6874 to (503.35, 491.9, 14.2) mm, rotated rx 0 ry 90 rz 0 deg; joints [-11.203, -27.757, 111.283, -15.221, -82.889, 50.925]
  Set speed (1000.0 mm/s)
  MoveL 6875 to (504.05, 491.9, 14.2) mm, rotated rx 0 ry 90 rz 0 deg; joints [-11.191, -27.743, 111.199, -15.21, -82.82, 50.942]
  Set speed (1000.0 mm/s)
  MoveL 6876 to (495.86, 492.33, 14.2) mm, rotated rx 0 ry 90 rz 0 deg; joints [-11.381, -27.892, 112.166, -15.376, -83.616, 50.744]
  Set speed (1000.0 mm/s)
  MoveL 6877 to (490.68, 490.68, 14.2) mm, rotated rx 0 ry 90 rz 0 deg; joints [-11.324, -27.987, 112.82, -15.303, -84.154, 50.59]
  Set speed (1000.0 mm/s)
  MoveL 6878 to (490.68, 490.68, 14.3) mm, rotated rx 0 ry 90 rz 0 deg; joints [-11.324, -27.997, 112.825, -15.303, -84.148, 50.591]
  Set speed (30.0 mm/s)
  Call Extruder(0.767)
  MoveL 6879 to (509.32, 509.32, 14.3) mm, rotated rx 0 ry 90 rz 0 deg; joints [-12.669, -27.577, 110.128, -16.733, -82, 51.368]
  MoveL 6880 to (509.44, 509.44, 14.3) mm, rotated rx 0 ry 90 rz 0 deg; joints [-12.677, -27.574, 110.109, -16.743, -81.986, 51.373]
  Set speed (120.0 mm/s)
  MoveL 6881 to (507.64, 503.72, 14.3) mm, rotated rx 0 ry 90 rz 0 deg; joints [-12.198, -27.636, 110.478, -16.247, -82.263, 51.226]
  Set speed (1000.0 mm/s)
  MoveL 6882 to (507.39, 502.51, 14.3) mm, rotated rx 0 ry 90 rz 0 deg; joints [-12.093, -27.646, 110.54, -16.14, -82.308, 51.199]
  Set speed (30.0 mm/s)
  Call Extruder(0.280)
  MoveL 6883 to (500.58, 509.32, 14.3) mm, rotated rx 0 ry 90 rz 0 deg; joints [-12.847, -27.749, 111.175, -16.88, -82.844, 51.133]
  Set speed (120.0 mm/s)
  MoveL 6884 to (499.42, 509.32, 14.3) mm, rotated rx 0 ry 90 rz 0 deg; joints [-12.872, -27.771, 111.313, -16.9, -82.956, 51.102]
  Set speed (30.0 mm/s)
  Call Extruder(0.360)
  MoveL 6885 to (490.68, 500.58, 14.3) mm, rotated rx 0 ry 90 rz 0 deg; joints [-12.247, -27.963, 112.581, -16.236, -83.97, 50.731]
  Set speed (120.0 mm/s)
  MoveL 6886 to (490.68, 499.42, 14.3) mm, rotated rx 0 ry 90 rz 0 deg; joints [-12.139, -27.967, 112.611, -16.127, -83.991, 50.714]
  Set speed (30.0 mm/s)
  Call Extruder(0.281)
  MoveL 6887 to (497.52, 492.58, 14.3) mm, rotated rx 0 ry 90 rz 0 deg; joints [-11.373, -27.872, 111.968, -15.374, -83.444, 50.791]
  MoveL 6888 to (497.64, 492.46, 14.3) mm, rotated rx 0 ry 90 rz 0 deg; joints [-11.36, -27.871, 111.957, -15.36, -83.434, 50.792]
  Set speed (120.0 mm/s)
  MoveL 6889 to (498.57, 491.53, 14.3) mm, rotated rx 0 ry 90 rz 0 deg; joints [-11.257, -27.857, 111.868, -15.259, -83.358, 50.802]
  Set speed (30.0 mm/s)
  Call Extruder(0.035)
  MoveL 6890 to (499.42, 490.68, 14.3) mm, rotated rx 0 ry 90 rz 0 deg; joints [-11.163, -27.845, 111.787, -15.166, -83.289, 50.81]
  Set speed (120.0 mm/s)
  MoveL 6891 to (500.58, 490.68, 14.3) mm, rotated rx 0 ry 90 rz 0 deg; joints [-11.141, -27.824, 111.648, -15.149, -83.175, 50.839]
  Set speed (30.0 mm/s)
  Call Extruder(0.005)
  MoveL 6892 to (500.69, 490.79, 14.3) mm, rotated rx 0 ry 90 rz 0 deg; joints [-11.15, -27.821, 111.632, -15.158, -83.162, 50.844]
  Set speed (120.0 mm/s)
  MoveL 6893 to (500.95, 492.33, 14.3) mm, rotated rx 0 ry 90 rz 0 deg; joints [-11.287, -27.811, 111.565, -15.297, -83.111, 50.873]
  Set speed (1000.0 mm/s)
  MoveL 6894 to (502.48, 492.58, 14.3) mm, rotated rx 0 ry 90 rz 0 deg; joints [-11.282, -27.781, 111.375, -15.297, -82.957, 50.915]
  Set speed (30.0 mm/s)
  Call Extruder(0.202)
  MoveL 6895 to (507.39, 497.49, 14.3) mm, rotated rx 0 ry 90 rz 0 deg; joints [-11.639, -27.667, 110.666, -15.677, -82.395, 51.116]
  Set speed (120.0 mm/s)
  MoveL 6896 to (508.05, 498.16, 14.3) mm, rotated rx 0 ry 90 rz 0 deg; joints [-11.687, -27.651, 110.57, -15.729, -82.319, 51.143]
  Set speed (30.0 mm/s)
  Call Extruder(0.052)
  MoveL 6897 to (509.32, 499.42, 14.3) mm, rotated rx 0 ry 90 rz 0 deg; joints [-11.777, -27.621, 110.386, -15.826, -82.174, 51.196]
  Set speed (120.0 mm/s)
  MoveL 6898 to (509.32, 500.58, 14.3) mm, rotated rx 0 ry 90 rz 0 deg; joints [-11.882, -27.616, 110.357, -15.932, -82.154, 51.216]
  Set speed (30.0 mm/s)
  Call Extruder(0.014)
  MoveL 6899 to (508.98, 500.91, 14.3) mm, rotated rx 0 ry 90 rz 0 deg; joints [-11.918, -27.621, 110.389, -15.968, -82.181, 51.213]
  Set speed (120.0 mm/s)
  MoveL 6900 to (507.64, 497.9, 14.3) mm, rotated rx 0 ry 90 rz 0 deg; joints [-11.671, -27.66, 110.626, -15.712, -82.363, 51.129]
  Set speed (1000.0 mm/s)
  MoveL 6901 to (507.64, 495.33, 14.3) mm, rotated rx 0 ry 90 rz 0 deg; joints [-11.438, -27.671, 110.689, -15.474, -82.406, 51.087]
  Set speed (1000.0 mm/s)
  MoveL 6902 to (509.32, 490.68, 14.3) mm, rotated rx 0 ry 90 rz 0 deg; joints [-10.985, -27.656, 110.598, -15.02, -82.319, 51.053]
  Set speed (30.0 mm/s)
  Call Extruder(0.767)
  MoveL 6903 to (490.68, 509.32, 14.3) mm, rotated rx 0 ry 90 rz 0 deg; joints [-13.056, -27.929, 112.35, -17.056, -83.802, 50.862]
  MoveL 6904 to (490.56, 509.44, 14.3) mm, rotated rx 0 ry 90 rz 0 deg; joints [-13.07, -27.931, 112.361, -17.07, -83.812, 50.861]
  Set speed (120.0 mm/s)
  MoveL 6905 to (503.48, 492.37, 14.3) mm, rotated rx 0 ry 90 rz 0 deg; joints [-11.244, -27.763, 111.261, -15.262, -82.863, 50.936]
  Set speed (1000.0 mm/s)
  MoveL 6906 to (503.41, 492.3, 14.3) mm, rotated rx 0 ry 90 rz 0 deg; joints [-11.239, -27.765, 111.271, -15.257, -82.871, 50.934]
  Set speed (15.0 mm/s)
  Call Extruder(0.010)
  MoveL 6907 to (503.41, 491.95, 14.3) mm, rotated rx 0 ry 90 rz 0 deg; joints [-11.207, -27.766, 111.279, -15.225, -82.876, 50.928]
  Call Extruder(0.035)
  MoveL 6908 to (503.41, 490.75, 14.3) mm, rotated rx 0 ry 90 rz 0 deg; joints [-11.097, -27.77, 111.307, -15.113, -82.896, 50.91]
  Call Extruder(0.010)
  MoveL 6909 to (503.41, 490.4, 14.3) mm, rotated rx 0 ry 90 rz 0 deg; joints [-11.065, -27.772, 111.316, -15.08, -82.902, 50.905]
  Call Extruder(0.007)
  MoveL 6910 to (503.76, 490.4, 14.3) mm, rotated rx 0 ry 90 rz 0 deg; joints [-11.059, -27.765, 111.274, -15.075, -82.868, 50.913]
  Call Extruder(0.170)
  MoveL 6911 to (509.6, 490.4, 14.3) mm, rotated rx 0 ry 90 rz 0 deg; joints [-10.955, -27.651, 110.571, -14.991, -82.296, 51.055]
  Call Extruder(0.144)
  MoveL 6912 to (509.6, 495.36, 14.3) mm, rotated rx 0 ry 90 rz 0 deg; joints [-11.404, -27.632, 110.453, -15.448, -82.215, 51.136]
  Call Extruder(0.056)
  MoveL 6913 to (507.67, 495.36, 14.3) mm, rotated rx 0 ry 90 rz 0 deg; joints [-11.44, -27.67, 110.685, -15.476, -82.403, 51.088]
  Call Extruder(0.073)
  MoveL 6914 to (507.67, 497.88, 14.3) mm, rotated rx 0 ry 90 rz 0 deg; joints [-11.668, -27.66, 110.623, -15.709, -82.361, 51.129]
  Call Extruder(0.056)
  MoveL 6915 to (509.6, 497.88, 14.3) mm, rotated rx 0 ry 90 rz 0 deg; joints [-11.632, -27.622, 110.391, -15.679, -82.173, 51.178]
  Call Extruder(0.086)
  MoveL 6916 to (509.6, 500.84, 14.3) mm, rotated rx 0 ry 90 rz 0 deg; joints [-11.9, -27.609, 110.316, -15.952, -82.123, 51.228]
  Call Extruder(0.010)
  MoveL 6917 to (509.6, 501.19, 14.3) mm, rotated rx 0 ry 90 rz 0 deg; joints [-11.932, -27.608, 110.307, -15.984, -82.117, 51.233]
  Call Extruder(0.007)
  MoveL 6918 to (509.25, 501.19, 14.3) mm, rotated rx 0 ry 90 rz 0 deg; joints [-11.939, -27.615, 110.349, -15.99, -82.151, 51.225]
  Call Extruder(0.036)
  MoveL 6919 to (508.02, 501.19, 14.3) mm, rotated rx 0 ry 90 rz 0 deg; joints [-11.962, -27.639, 110.498, -16.008, -82.27, 51.193]
  Call Extruder(0.010)
  MoveL 6920 to (507.67, 501.19, 14.3) mm, rotated rx 0 ry 90 rz 0 deg; joints [-11.969, -27.646, 110.54, -16.014, -82.304, 51.184]
  Call Extruder(0.007)
  MoveL 6921 to (507.67, 501.54, 14.3) mm, rotated rx 0 ry 90 rz 0 deg; joints [-12, -27.645, 110.531, -16.046, -82.298, 51.19]
  Call Extruder(0.063)
  MoveL 6922 to (507.67, 503.69, 14.3) mm, rotated rx 0 ry 90 rz 0 deg; joints [-12.195, -27.636, 110.476, -16.244, -82.26, 51.226]
  Call Extruder(0.056)
  MoveL 6923 to (509.6, 503.7, 14.3) mm, rotated rx 0 ry 90 rz 0 deg; joints [-12.157, -27.597, 110.243, -16.214, -82.073, 51.276]
  Call Extruder(0.172)
  MoveL 6924 to (509.6, 509.6, 14.3) mm, rotated rx 0 ry 90 rz 0 deg; joints [-12.688, -27.57, 110.086, -16.754, -81.968, 51.38]
  Call Extruder(0.559)
  MoveL 6925 to (490.4, 509.6, 14.3) mm, rotated rx 0 ry 90 rz 0 deg; joints [-13.088, -27.933, 112.375, -17.087, -83.824, 50.859]
  MoveL 6926 to (490.4, 490.4, 14.3) mm, rotated rx 0 ry 90 rz 0 deg; joints [-11.303, -28.003, 112.865, -15.281, -84.181, 50.581]
  Call Extruder(0.148)
  MoveL 6927 to (495.48, 490.4, 14.3) mm, rotated rx 0 ry 90 rz 0 deg; joints [-11.209, -27.916, 112.262, -15.201, -83.68, 50.708]
  Call Extruder(0.010)
  MoveL 6928 to (495.83, 490.4, 14.3) mm, rotated rx 0 ry 90 rz 0 deg; joints [-11.202, -27.91, 112.221, -15.195, -83.646, 50.717]
  Call Extruder(0.007)
  MoveL 6929 to (495.83, 490.75, 14.3) mm, rotated rx 0 ry 90 rz 0 deg; joints [-11.235, -27.909, 112.212, -15.228, -83.64, 50.722]
  Call Extruder(0.035)
  MoveL 6930 to (495.83, 491.95, 14.3) mm, rotated rx 0 ry 90 rz 0 deg; joints [-11.346, -27.905, 112.184, -15.341, -83.62, 50.739]
  Call Extruder(0.010)
  MoveL 6931 to (495.83, 492.3, 14.3) mm, rotated rx 0 ry 90 rz 0 deg; joints [-11.379, -27.903, 112.176, -15.374, -83.614, 50.744]
  Call Extruder(0.007)
  MoveL 6932 to (496.18, 492.3, 14.3) mm, rotated rx 0 ry 90 rz 0 deg; joints [-11.372, -27.897, 112.134, -15.368, -83.579, 50.753]
  Call Extruder(0.061)
  MoveL 6933 to (498.29, 492.3, 14.3) mm, rotated rx 0 ry 90 rz 0 deg; joints [-11.333, -27.859, 111.883, -15.335, -83.373, 50.806]
  Call Extruder(0.055)
  MoveL 6934 to (498.29, 490.4, 14.3) mm, rotated rx 0 ry 90 rz 0 deg; joints [-11.157, -27.866, 111.928, -15.157, -83.405, 50.778]
  Call Extruder(0.078)
  MoveL 6935 to (500.97, 490.4, 14.3) mm, rotated rx 0 ry 90 rz 0 deg; joints [-11.109, -27.817, 111.607, -15.117, -83.141, 50.845]
  Call Extruder(0.055)
  MoveL 6936 to (500.98, 492.3, 14.3) mm, rotated rx 0 ry 90 rz 0 deg; joints [-11.284, -27.81, 111.562, -15.294, -83.109, 50.873]
  Call Extruder(0.061)
  MoveL 6937 to (503.06, 492.3, 14.3) mm, rotated rx 0 ry 90 rz 0 deg; joints [-11.245, -27.771, 111.313, -15.262, -82.905, 50.925]
  Call Extruder(0.007)
  MoveL 6938 to (503.41, 492.3, 14.3) mm, rotated rx 0 ry 90 rz 0 deg; joints [-11.239, -27.765, 111.271, -15.257, -82.871, 50.934]
  Set speed (120.0 mm/s)
  MoveL 6939 to (503.41, 491.95, 14.3) mm, rotated rx 0 ry 90 rz 0 deg; joints [-11.207, -27.766, 111.279, -15.225, -82.876, 50.928]
  Set speed (1000.0 mm/s)
  MoveL 6940 to (503.41, 491.9, 14.3) mm, rotated rx 0 ry 90 rz 0 deg; joints [-11.202, -27.766, 111.28, -15.22, -82.877, 50.928]
  Set speed (1000.0 mm/s)
  MoveL 6941 to (504.11, 491.9, 14.3) mm, rotated rx 0 ry 90 rz 0 deg; joints [-11.19, -27.753, 111.196, -15.209, -82.809, 50.945]
  Set speed (1000.0 mm/s)
  MoveL 6942 to (495.8, 492.33, 14.3) mm, rotated rx 0 ry 90 rz 0 deg; joints [-11.382, -27.904, 112.178, -15.377, -83.616, 50.744]
  Set speed (1000.0 mm/s)
  MoveL 6943 to (490.68, 490.68, 14.3) mm, rotated rx 0 ry 90 rz 0 deg; joints [-11.324, -27.997, 112.825, -15.303, -84.148, 50.591]
  Set speed (1000.0 mm/s)
  MoveL 6944 to (490.68, 490.68, 14.4) mm, rotated rx 0 ry 90 rz 0 deg; joints [-11.324, -28.008, 112.831, -15.303, -84.143, 50.593]
  Set speed (30.0 mm/s)
  Call Extruder(0.767)
  MoveL 6945 to (509.32, 509.32, 14.4) mm, rotated rx 0 ry 90 rz 0 deg; joints [-12.669, -27.588, 110.133, -16.734, -81.995, 51.369]
  MoveL 6946 to (509.44, 509.44, 14.4) mm, rotated rx 0 ry 90 rz 0 deg; joints [-12.677, -27.585, 110.115, -16.743, -81.981, 51.375]
  Set speed (120.0 mm/s)
  MoveL 6947 to (507.64, 503.78, 14.4) mm, rotated rx 0 ry 90 rz 0 deg; joints [-12.203, -27.646, 110.482, -16.252, -82.256, 51.229]
  Set speed (1000.0 mm/s)
  MoveL 6948 to (507.39, 502.51, 14.4) mm, rotated rx 0 ry 90 rz 0 deg; joints [-12.093, -27.657, 110.545, -16.14, -82.303, 51.201]
  Set speed (30.0 mm/s)
  Call Extruder(0.280)
  MoveL 6949 to (500.58, 509.32, 14.4) mm, rotated rx 0 ry 90 rz 0 deg; joints [-12.847, -27.76, 111.18, -16.88, -82.839, 51.135]
  Set speed (120.0 mm/s)
  MoveL 6950 to (499.42, 509.32, 14.4) mm, rotated rx 0 ry 90 rz 0 deg; joints [-12.872, -27.782, 111.318, -16.9, -82.951, 51.104]
  Set speed (30.0 mm/s)
  Call Extruder(0.360)
  MoveL 6951 to (490.68, 500.58, 14.4) mm, rotated rx 0 ry 90 rz 0 deg; joints [-12.247, -27.973, 112.586, -16.236, -83.965, 50.732]
  Set speed (120.0 mm/s)
  MoveL 6952 to (490.68, 499.42, 14.4) mm, rotated rx 0 ry 90 rz 0 deg; joints [-12.139, -27.977, 112.616, -16.127, -83.986, 50.715]
  Set speed (30.0 mm/s)
  Call Extruder(0.281)
  MoveL 6953 to (497.52, 492.58, 14.4) mm, rotated rx 0 ry 90 rz 0 deg; joints [-11.373, -27.883, 111.973, -15.374, -83.438, 50.792]
  MoveL 6954 to (497.64, 492.46, 14.4) mm, rotated rx 0 ry 90 rz 0 deg; joints [-11.36, -27.881, 111.962, -15.36, -83.428, 50.794]
  Set speed (120.0 mm/s)
  MoveL 6955 to (498.51, 491.59, 14.4) mm, rotated rx 0 ry 90 rz 0 deg; joints [-11.263, -27.869, 111.879, -15.265, -83.358, 50.803]
  Set speed (30.0 mm/s)
  Call Extruder(0.037)
  MoveL 6956 to (499.42, 490.68, 14.4) mm, rotated rx 0 ry 90 rz 0 deg; joints [-11.163, -27.855, 111.792, -15.166, -83.284, 50.812]
  Set speed (120.0 mm/s)
  MoveL 6957 to (500.58, 490.68, 14.4) mm, rotated rx 0 ry 90 rz 0 deg; joints [-11.142, -27.834, 111.653, -15.149, -83.17, 50.841]
  Set speed (30.0 mm/s)
  Call Extruder(0.007)
  MoveL 6958 to (500.76, 490.86, 14.4) mm, rotated rx 0 ry 90 rz 0 deg; joints [-11.155, -27.83, 111.628, -15.163, -83.149, 50.848]
  Set speed (120.0 mm/s)
  MoveL 6959 to (501.01, 492.33, 14.4) mm, rotated rx 0 ry 90 rz 0 deg; joints [-11.285, -27.82, 111.562, -15.296, -83.1, 50.876]
  Set speed (1000.0 mm/s)
  MoveL 6960 to (502.48, 492.58, 14.4) mm, rotated rx 0 ry 90 rz 0 deg; joints [-11.282, -27.792, 111.381, -15.297, -82.952, 50.916]
  Set speed (30.0 mm/s)
  Call Extruder(0.202)
  MoveL 6961 to (507.39, 497.49, 14.4) mm, rotated rx 0 ry 90 rz 0 deg; joints [-11.639, -27.678, 110.671, -15.678, -82.389, 51.117]
  Set speed (120.0 mm/s)
  MoveL 6962 to (508, 498.1, 14.4) mm, rotated rx 0 ry 90 rz 0 deg; joints [-11.682, -27.663, 110.583, -15.724, -82.32, 51.142]
  Set speed (30.0 mm/s)
  Call Extruder(0.054)
  MoveL 6963 to (509.32, 499.42, 14.4) mm, rotated rx 0 ry 90 rz 0 deg; joints [-11.777, -27.631, 110.391, -15.826, -82.169, 51.198]
  Set speed (120.0 mm/s)
  MoveL 6964 to (509.32, 500.58, 14.4) mm, rotated rx 0 ry 90 rz 0 deg; joints [-11.882, -27.626, 110.362, -15.932, -82.149, 51.217]
  Set speed (30.0 mm/s)
  Call Extruder(0.016)
  MoveL 6965 to (508.93, 500.97, 14.4) mm, rotated rx 0 ry 90 rz 0 deg; joints [-11.924, -27.633, 110.399, -15.974, -82.18, 51.214]
  Set speed (120.0 mm/s)
  MoveL 6966 to (507.65, 497.85, 14.4) mm, rotated rx 0 ry 90 rz 0 deg; joints [-11.666, -27.671, 110.632, -15.706, -82.359, 51.129]
  Set speed (1000.0 mm/s)
  MoveL 6967 to (507.64, 495.27, 14.4) mm, rotated rx 0 ry 90 rz 0 deg; joints [-11.432, -27.682, 110.696, -15.469, -82.402, 51.087]
  Set speed (1000.0 mm/s)
  MoveL 6968 to (509.32, 490.68, 14.4) mm, rotated rx 0 ry 90 rz 0 deg; joints [-10.985, -27.666, 110.603, -15.021, -82.313, 51.054]
  Set speed (30.0 mm/s)
  Call Extruder(0.767)
  MoveL 6969 to (490.68, 509.32, 14.4) mm, rotated rx 0 ry 90 rz 0 deg; joints [-13.056, -27.94, 112.355, -17.056, -83.797, 50.864]
  MoveL 6970 to (490.56, 509.44, 14.4) mm, rotated rx 0 ry 90 rz 0 deg; joints [-13.07, -27.941, 112.366, -17.07, -83.806, 50.862]
  Set speed (120.0 mm/s)
  MoveL 6971 to (503.55, 492.37, 14.4) mm, rotated rx 0 ry 90 rz 0 deg; joints [-11.243, -27.772, 111.258, -15.262, -82.851, 50.94]
  Set speed (1000.0 mm/s)
  MoveL 6972 to (503.48, 492.3, 14.4) mm, rotated rx 0 ry 90 rz 0 deg; joints [-11.238, -27.774, 111.268, -15.256, -82.859, 50.937]
  Set speed (15.0 mm/s)
  Call Extruder(0.010)
  MoveL 6973 to (503.48, 491.95, 14.4) mm, rotated rx 0 ry 90 rz 0 deg; joints [-11.206, -27.775, 111.276, -15.224, -82.865, 50.931]
  Call Extruder(0.035)
  MoveL 6974 to (503.47, 490.75, 14.4) mm, rotated rx 0 ry 90 rz 0 deg; joints [-11.096, -27.78, 111.305, -15.112, -82.885, 50.913]
  Call Extruder(0.010)
  MoveL 6975 to (503.47, 490.4, 14.4) mm, rotated rx 0 ry 90 rz 0 deg; joints [-11.064, -27.781, 111.313, -15.08, -82.891, 50.908]
  Call Extruder(0.007)
  MoveL 6976 to (503.82, 490.4, 14.4) mm, rotated rx 0 ry 90 rz 0 deg; joints [-11.057, -27.774, 111.271, -15.074, -82.856, 50.916]
  Call Extruder(0.168)
  MoveL 6977 to (509.6, 490.4, 14.4) mm, rotated rx 0 ry 90 rz 0 deg; joints [-10.955, -27.662, 110.576, -14.991, -82.29, 51.057]
  Call Extruder(0.143)
  MoveL 6978 to (509.6, 495.3, 14.4) mm, rotated rx 0 ry 90 rz 0 deg; joints [-11.399, -27.643, 110.459, -15.442, -82.211, 51.136]
  Call Extruder(0.056)
  MoveL 6979 to (507.67, 495.3, 14.4) mm, rotated rx 0 ry 90 rz 0 deg; joints [-11.435, -27.681, 110.692, -15.471, -82.399, 51.088]
  Call Extruder(0.063)
  MoveL 6980 to (507.67, 497.47, 14.4) mm, rotated rx 0 ry 90 rz 0 deg; joints [-11.631, -27.672, 110.638, -15.671, -82.362, 51.124]
  Call Extruder(0.010)
  MoveL 6981 to (507.67, 497.82, 14.4) mm, rotated rx 0 ry 90 rz 0 deg; joints [-11.663, -27.671, 110.629, -15.703, -82.357, 51.13]
  Call Extruder(0.007)
  MoveL 6982 to (508.02, 497.82, 14.4) mm, rotated rx 0 ry 90 rz 0 deg; joints [-11.657, -27.664, 110.587, -15.698, -82.322, 51.138]
  Call Extruder(0.046)
  MoveL 6983 to (509.6, 497.82, 14.4) mm, rotated rx 0 ry 90 rz 0 deg; joints [-11.627, -27.632, 110.397, -15.674, -82.169, 51.178]
  Call Extruder(0.100)
  MoveL 6984 to (509.6, 501.25, 14.4) mm, rotated rx 0 ry 90 rz 0 deg; joints [-11.937, -27.618, 110.311, -15.99, -82.11, 51.236]
  Call Extruder(0.046)
  MoveL 6985 to (508.02, 501.25, 14.4) mm, rotated rx 0 ry 90 rz 0 deg; joints [-11.967, -27.65, 110.501, -16.014, -82.264, 51.195]
  Call Extruder(0.010)
  MoveL 6986 to (507.67, 501.25, 14.4) mm, rotated rx 0 ry 90 rz 0 deg; joints [-11.974, -27.657, 110.543, -16.019, -82.298, 51.186]
  Call Extruder(0.007)
  MoveL 6987 to (507.67, 501.6, 14.4) mm, rotated rx 0 ry 90 rz 0 deg; joints [-12.005, -27.655, 110.535, -16.051, -82.292, 51.192]
  Call Extruder(0.063)
  MoveL 6988 to (507.67, 503.75, 14.4) mm, rotated rx 0 ry 90 rz 0 deg; joints [-12.2, -27.646, 110.479, -16.249, -82.254, 51.229]
  Call Extruder(0.056)
  MoveL 6989 to (509.6, 503.75, 14.4) mm, rotated rx 0 ry 90 rz 0 deg; joints [-12.163, -27.607, 110.247, -16.219, -82.067, 51.279]
  Call Extruder(0.170)
